(* Logix 5000 project; controller Comas_L4 vendor 1 type 14 code 193 rev 30.11; software revision 30.02; part 7 of 12 *)

        [27].Comas.Tete.Cam_Axe_Vertical[5].Master := 66.0, [27].Comas.Tete.Cam_Axe_Vertical[5].Slave := 14.0, [27].Comas.Tete.Cam_Axe_Vertical[5].SegmentType := 1, [27].Comas.Tete.Cam_Axe_Vertical[6].Master := 86.0, [27].Comas.Tete.Cam_Axe_Vertical[7].Master := 95.0, [27].Comas.Tete.Longueur_Cam_Axe_H := 8, [27].Comas.Tete.Offset_Vertical_Gauche := 38.0, [27].Comas.Tete.Offset_Horizontal_Gauche := 95.0, [27].Comas.Tete.Cam_Axe_Horizontal_Pan.B.x := 1.0, [27].Comas.Tete.Cam_Axe_Horizontal_Pan.C.x := 10.0, [27].Comas.Tete.Cam_Axe_Horizontal_Pan.C.y := 5.0, [27].Comas.Tete.Cam_Axe_Horizontal_Pan.D.x := 30.0, [27].Comas.Tete.Cam_Axe_Horizontal_Pan.D.y := 30.0, [27].Comas.Tete.Cam_Axe_Horizontal_Pan.E.x := 10.0, [27].Comas.Tete.Cam_Axe_Horizontal_Pan.E.y := 5.0, [27].Comas.Tete.Cam_Axe_Horizontal_Pan.F.x := 10.0, [27].Comas.Tete.Cam_Axe_Horizontal_Pan.G.x := 10.0, [27].Comas.Tete.Cam_Axe_Horizontal_Pan.G.y := -10.0, [27].Comas.Tete.Cam_Axe_Vertical_Pan.K.y := 2.0, [27].Comas.Tete.Cam_Axe_Vertical_Pan.L.x := 14.0, [27].Comas.Tete.Cam_Axe_Vertical_Pan.L.y := 15.0, [27].Comas.Tete.Cam_Axe_Vertical_Pan.M.x := 5.0, [27].Comas.Tete.Cam_Axe_Vertical_Pan.M.y := 14.0, [27].Comas.Tete.Cam_Axe_Vertical_Pan.N.x := 15.0, [27].Comas.Tete.Offset_Vertical_Droit := 45.0, [27].Comas.Tete.Offset_Horizontal_Droit := 95.0, [27].Comas.Pompe.Start_Cam_Logique_Avance := 1.0, [27].Comas.Pompe.Stop_Cam_Logique_Avance := 14.0, [27].Comas.Pompe.Start_Cam_Logique_Recul := 16.0, [27].Comas.Pompe.Stop_Cam_Logique_Recul := 31.0, [27].Comas.Pompe.Consigne_Vitesse_Avance := 13.2, [27].Comas.Pompe.Consigne_Acc_Dec_Avance := 40.0, [27].Comas.Pompe.Consigne_Jerk_Avance := 100.0, [27].Comas.Pompe.Consigne_Acc_Dec_Recul := 40.0, [27].Comas.Pompe.Consigne_Jerk_Recul := 100.0, [27].Comas.Pompe.Points_Pan.O.x := -10.0, [27].Comas.Pompe.Points_Pan.Q.x := 13.0, [27].Comas.Pompe.Points_Pan.S.x := -25.0, [27].Comas.Pompe.Points_Pan.U.x := 15.0, [27].Comas.Pompe.Reserve_Bool1 := 1, [27].Comas.Rouleaux.Syncho_Pompe := 1, [27].Comas.Rouleaux.Consigne_Vitesse := 30.0, [27].Comas.Rouleaux.Consigne_Acc_Dec := 40.0, [27].Comas.Rouleaux.Consigne_Jerk := 100.0, [27].Comas.Rouleaux.Reserve_Real1 := -20.0, [27].Comas.Coupe_Fil.Activation := 1, [27].Comas.Coupe_Fil.Start_Cam_Logique_Virtuelle := 11.0, [27].Comas.Coupe_Fil.Stop_Cam_Logique_Virtuelle := 21.0, [27].Comas.Coupe_Fil.Consigne_Vitesse_Virtuelle := 250.0, [27].Comas.Coupe_Fil.Consigne_Acc_Dec_Virtuelle := 1000.0, [27].Comas.Coupe_Fil.Consigne_Jerk_Virtuelle := 50.0, [27].Comas.Coupe_Fil.Cam_Axe[0].SegmentType := 1, [27].Comas.Coupe_Fil.Cam_Axe[1].Master := 180.0, [27].Comas.Coupe_Fil.Cam_Axe[1].Slave := 180.0, [27].Comas.Coupe_Fil.Cam_Axe[2].Master := 250.0, [27].Comas.Coupe_Fil.Cam_Axe[2].Slave := 200.0, [27].Comas.Coupe_Fil.Cam_Axe[2].SegmentType := 1, [27].Comas.Coupe_Fil.Cam_Axe[3].Master := 360.0, [27].Comas.Coupe_Fil.Cam_Axe[3].Slave := 360.0, [27].Comas.Coupe_Fil.Cam_Axe[3].SegmentType := 1,
        [27].Comas.Coupe_Fil.Cam_Axe[4].SegmentType := 1, [27].Comas.Coupe_Fil.Points_Pan.W.x := -40.0, [27].Comas.Coupe_Fil.Reserve_Bool1 := 1, [27].Comas.Consigne_Vitesse_Manu_mm := 2.0, [27].Comas.Consigne_Acc_Decc_Manu_mm := 10.0, [27].Comas.Consigne_Jerk_Manu := 100.0, [27].Comas.Activation_Cam_Auto := 1, [27].Comas.Distance_CPT_Presence_Produit := 520, [27].Comas.Consigne_Vitesse_Manu_Tour := 10.0, [27].Comas.Consigne_Acc_Decc_Manu_Tour := 10.0, [27].Comas.Mode_Decoreuse_Cam_Logique := 1, [27].Comas.Reserve_Real3 := 1.0, [27].Comas.Reserve_Real4 := 1.0, [27].Comas.Reserve_Real5 := 5.0, [27].Comas.Reserve_Real6 := 200.0, [27].Reserve_Real2 := 200.0, [27].Reserve_Real3 := 10.0, [28].Name := 'Galette framboise', [28].Comas.Pas_Machine := 78, [28].Comas.Came_Maitre[1].Master := 78.0, [28].Comas.Came_Maitre[1].Slave := 78.0, [28].Comas.Longueur_Came_Maitre := 2, [28].Comas.Tete.Stop_Cam_Logique_Degagement := 10.0, [28].Comas.Tete.Position_Degagement_H := 50.0, [28].Comas.Tete.Position_Degagement_V := 37.0, [28].Comas.Tete.Hauteur_Tete := -23, [28].Comas.Tete.Cam_Axe_Horizontal[1].Master := 1.0, [28].Comas.Tete.Cam_Axe_Horizontal[2].Master := 11.0, [28].Comas.Tete.Cam_Axe_Horizontal[2].Slave := -3.0, [28].Comas.Tete.Cam_Axe_Horizontal[3].Master := 41.0, [28].Comas.Tete.Cam_Axe_Horizontal[3].Slave := -6.0, [28].Comas.Tete.Cam_Axe_Horizontal[3].SegmentType := 1, [28].Comas.Tete.Cam_Axe_Horizontal[4].Master := 53.0, [28].Comas.Tete.Cam_Axe_Horizontal[4].Slave := 4.0, [28].Comas.Tete.Cam_Axe_Horizontal[4].SegmentType := 1, [28].Comas.Tete.Cam_Axe_Horizontal[5].Master := 63.0, [28].Comas.Tete.Cam_Axe_Horizontal[5].Slave := 9.0, [28].Comas.Tete.Cam_Axe_Horizontal[5].SegmentType := 1, [28].Comas.Tete.Cam_Axe_Horizontal[6].Master := 73.0, [28].Comas.Tete.Cam_Axe_Horizontal[6].Slave := 4.0, [28].Comas.Tete.Cam_Axe_Horizontal[6].SegmentType := 1, [28].Comas.Tete.Cam_Axe_Horizontal[7].Master := 78.0, [28].Comas.Tete.Cam_Axe_Vertical[1].Master := 1.0, [28].Comas.Tete.Cam_Axe_Vertical[2].Master := 11.0, [28].Comas.Tete.Cam_Axe_Vertical[3].Master := 41.0, [28].Comas.Tete.Cam_Axe_Vertical[3].SegmentType := 1, [28].Comas.Tete.Cam_Axe_Vertical[4].Master := 53.0, [28].Comas.Tete.Cam_Axe_Vertical[4].Slave := 15.0, [28].Comas.Tete.Cam_Axe_Vertical[5].Master := 63.0, [28].Comas.Tete.Cam_Axe_Vertical[5].Slave := 20.0, [28].Comas.Tete.Cam_Axe_Vertical[5].SegmentType := 1, [28].Comas.Tete.Cam_Axe_Vertical[6].Master := 73.0, [28].Comas.Tete.Cam_Axe_Vertical[6].Slave := 12.0, [28].Comas.Tete.Cam_Axe_Vertical[6].SegmentType := 1, [28].Comas.Tete.Cam_Axe_Vertical[7].Master := 78.0, [28].Comas.Tete.Longueur_Cam_Axe_H := 8, [28].Comas.Tete.Offset_Vertical_Gauche := 38.0, [28].Comas.Tete.Offset_Horizontal_Gauche := 94.0, [28].Comas.Tete.Cam_Axe_Horizontal_Pan.B.x := 1.0, [28].Comas.Tete.Cam_Axe_Horizontal_Pan.C.x := 10.0,
        [28].Comas.Tete.Cam_Axe_Horizontal_Pan.C.y := -3.0, [28].Comas.Tete.Cam_Axe_Horizontal_Pan.D.x := 30.0, [28].Comas.Tete.Cam_Axe_Horizontal_Pan.D.y := 5.0, [28].Comas.Tete.Cam_Axe_Horizontal_Pan.E.x := 12.0, [28].Comas.Tete.Cam_Axe_Horizontal_Pan.E.y := 10.0, [28].Comas.Tete.Cam_Axe_Horizontal_Pan.F.x := 10.0, [28].Comas.Tete.Cam_Axe_Horizontal_Pan.F.y := 5.0, [28].Comas.Tete.Cam_Axe_Horizontal_Pan.G.x := 10.0, [28].Comas.Tete.Cam_Axe_Horizontal_Pan.G.y := -5.0, [28].Comas.Tete.Cam_Axe_Vertical_Pan.L.y := 15.0, [28].Comas.Tete.Cam_Axe_Vertical_Pan.M.y := 20.0, [28].Comas.Tete.Cam_Axe_Vertical_Pan.N.y := 12.0, [28].Comas.Tete.Offset_Vertical_Droit := 45.0, [28].Comas.Tete.Offset_Horizontal_Droit := 94.0, [28].Comas.Tete.Reserve_Real1 := -8.0, [28].Comas.Pompe.Start_Cam_Logique_Avance := 1.0, [28].Comas.Pompe.Stop_Cam_Logique_Avance := 14.0, [28].Comas.Pompe.Start_Cam_Logique_Recul := 41.0, [28].Comas.Pompe.Stop_Cam_Logique_Recul := 41.0, [28].Comas.Pompe.Consigne_Vitesse_Avance := 18.2, [28].Comas.Pompe.Consigne_Acc_Dec_Avance := 40.0, [28].Comas.Pompe.Consigne_Jerk_Avance := 100.0, [28].Comas.Pompe.Consigne_Acc_Dec_Recul := 40.0, [28].Comas.Pompe.Consigne_Jerk_Recul := 100.0, [28].Comas.Pompe.Points_Pan.O.x := -10.0, [28].Comas.Pompe.Points_Pan.Q.x := 13.0, [28].Comas.Pompe.Reserve_Bool1 := 1, [28].Comas.Rouleaux.Syncho_Pompe := 1, [28].Comas.Rouleaux.Consigne_Vitesse := 25.0, [28].Comas.Rouleaux.Consigne_Acc_Dec := 40.0, [28].Comas.Rouleaux.Consigne_Jerk := 100.0, [28].Comas.Rouleaux.Reserve_Real1 := -10.0, [28].Comas.Coupe_Fil.Activation := 1, [28].Comas.Coupe_Fil.Start_Cam_Logique_Virtuelle := 18.0, [28].Comas.Coupe_Fil.Stop_Cam_Logique_Virtuelle := 28.0, [28].Comas.Coupe_Fil.Consigne_Vitesse_Virtuelle := 400.0, [28].Comas.Coupe_Fil.Consigne_Acc_Dec_Virtuelle := 1200.0, [28].Comas.Coupe_Fil.Consigne_Jerk_Virtuelle := 50.0, [28].Comas.Coupe_Fil.Cam_Axe[0].SegmentType := 1, [28].Comas.Coupe_Fil.Cam_Axe[1].Master := 180.0, [28].Comas.Coupe_Fil.Cam_Axe[1].Slave := 180.0, [28].Comas.Coupe_Fil.Cam_Axe[2].Master := 250.0, [28].Comas.Coupe_Fil.Cam_Axe[2].Slave := 200.0, [28].Comas.Coupe_Fil.Cam_Axe[2].SegmentType := 1, [28].Comas.Coupe_Fil.Cam_Axe[3].Master := 360.0, [28].Comas.Coupe_Fil.Cam_Axe[3].Slave := 360.0, [28].Comas.Coupe_Fil.Cam_Axe[3].SegmentType := 1, [28].Comas.Coupe_Fil.Cam_Axe[4].SegmentType := 1, [28].Comas.Coupe_Fil.Points_Pan.W.x := -35.0, [28].Comas.Coupe_Fil.Reserve_Bool1 := 1, [28].Comas.Consigne_Vitesse_Manu_mm := 2.0, [28].Comas.Consigne_Acc_Decc_Manu_mm := 10.0, [28].Comas.Consigne_Jerk_Manu := 100.0, [28].Comas.Activation_Cam_Auto := 1, [28].Comas.Distance_CPT_Presence_Produit := 520, [28].Comas.Consigne_Vitesse_Manu_Tour := 10.0, [28].Comas.Consigne_Acc_Decc_Manu_Tour := 10.0, [28].Comas.Mode_Decoreuse_Cam_Logique := 1, [28].Comas.Reserve_Real3 := 1.0, [28].Comas.Reserve_Real4 := 1.0,
        [28].Comas.Reserve_Real5 := 5.0, [28].Comas.Reserve_Real6 := 200.0, [28].Reserve_Real2 := 200.0, [28].Reserve_Real3 := 10.0, [29].Name := 'Galette orange', [29].Comas.Pas_Machine := 78, [29].Comas.Came_Maitre[1].Master := 78.0, [29].Comas.Came_Maitre[1].Slave := 78.0, [29].Comas.Longueur_Came_Maitre := 2, [29].Comas.Tete.Stop_Cam_Logique_Degagement := 10.0, [29].Comas.Tete.Position_Degagement_H := 50.0, [29].Comas.Tete.Position_Degagement_V := 37.0, [29].Comas.Tete.Hauteur_Tete := -24, [29].Comas.Tete.Cam_Axe_Horizontal[1].Master := 1.0, [29].Comas.Tete.Cam_Axe_Horizontal[2].Master := 11.0, [29].Comas.Tete.Cam_Axe_Horizontal[2].Slave := -3.0, [29].Comas.Tete.Cam_Axe_Horizontal[3].Master := 41.0, [29].Comas.Tete.Cam_Axe_Horizontal[3].Slave := -6.0, [29].Comas.Tete.Cam_Axe_Horizontal[3].SegmentType := 1, [29].Comas.Tete.Cam_Axe_Horizontal[4].Master := 53.0, [29].Comas.Tete.Cam_Axe_Horizontal[4].Slave := 4.0, [29].Comas.Tete.Cam_Axe_Horizontal[4].SegmentType := 1, [29].Comas.Tete.Cam_Axe_Horizontal[5].Master := 63.0, [29].Comas.Tete.Cam_Axe_Horizontal[5].Slave := 9.0, [29].Comas.Tete.Cam_Axe_Horizontal[5].SegmentType := 1, [29].Comas.Tete.Cam_Axe_Horizontal[6].Master := 73.0, [29].Comas.Tete.Cam_Axe_Horizontal[6].Slave := 4.0, [29].Comas.Tete.Cam_Axe_Horizontal[6].SegmentType := 1, [29].Comas.Tete.Cam_Axe_Horizontal[7].Master := 78.0, [29].Comas.Tete.Cam_Axe_Vertical[1].Master := 1.0, [29].Comas.Tete.Cam_Axe_Vertical[2].Master := 11.0, [29].Comas.Tete.Cam_Axe_Vertical[3].Master := 41.0, [29].Comas.Tete.Cam_Axe_Vertical[3].SegmentType := 1, [29].Comas.Tete.Cam_Axe_Vertical[4].Master := 53.0, [29].Comas.Tete.Cam_Axe_Vertical[4].Slave := 15.0, [29].Comas.Tete.Cam_Axe_Vertical[5].Master := 63.0, [29].Comas.Tete.Cam_Axe_Vertical[5].Slave := 25.0, [29].Comas.Tete.Cam_Axe_Vertical[5].SegmentType := 1, [29].Comas.Tete.Cam_Axe_Vertical[6].Master := 73.0, [29].Comas.Tete.Cam_Axe_Vertical[6].Slave := 12.0, [29].Comas.Tete.Cam_Axe_Vertical[6].SegmentType := 1, [29].Comas.Tete.Cam_Axe_Vertical[7].Master := 78.0, [29].Comas.Tete.Longueur_Cam_Axe_H := 8, [29].Comas.Tete.Offset_Vertical_Gauche := 38.0, [29].Comas.Tete.Offset_Horizontal_Gauche := 94.0, [29].Comas.Tete.Cam_Axe_Horizontal_Pan.B.x := 1.0, [29].Comas.Tete.Cam_Axe_Horizontal_Pan.C.x := 10.0, [29].Comas.Tete.Cam_Axe_Horizontal_Pan.C.y := -3.0, [29].Comas.Tete.Cam_Axe_Horizontal_Pan.D.x := 30.0, [29].Comas.Tete.Cam_Axe_Horizontal_Pan.D.y := 5.0, [29].Comas.Tete.Cam_Axe_Horizontal_Pan.E.x := 12.0, [29].Comas.Tete.Cam_Axe_Horizontal_Pan.E.y := 10.0, [29].Comas.Tete.Cam_Axe_Horizontal_Pan.F.x := 10.0, [29].Comas.Tete.Cam_Axe_Horizontal_Pan.F.y := 5.0, [29].Comas.Tete.Cam_Axe_Horizontal_Pan.G.x := 10.0, [29].Comas.Tete.Cam_Axe_Horizontal_Pan.G.y := -5.0, [29].Comas.Tete.Cam_Axe_Vertical_Pan.L.y := 15.0, [29].Comas.Tete.Cam_Axe_Vertical_Pan.M.y := 25.0, [29].Comas.Tete.Cam_Axe_Vertical_Pan.N.y := 12.0, [29].Comas.Tete.Offset_Vertical_Droit := 45.0,
        [29].Comas.Tete.Offset_Horizontal_Droit := 94.0, [29].Comas.Tete.Reserve_Real1 := -8.0, [29].Comas.Pompe.Start_Cam_Logique_Avance := 16.0, [29].Comas.Pompe.Stop_Cam_Logique_Avance := 29.0, [29].Comas.Pompe.Start_Cam_Logique_Recul := 41.0, [29].Comas.Pompe.Stop_Cam_Logique_Recul := 41.0, [29].Comas.Pompe.Consigne_Vitesse_Avance := 21.6, [29].Comas.Pompe.Consigne_Acc_Dec_Avance := 40.0, [29].Comas.Pompe.Consigne_Jerk_Avance := 100.0, [29].Comas.Pompe.Consigne_Acc_Dec_Recul := 40.0, [29].Comas.Pompe.Consigne_Jerk_Recul := 100.0, [29].Comas.Pompe.Points_Pan.O.x := 5.0, [29].Comas.Pompe.Points_Pan.Q.x := 13.0, [29].Comas.Pompe.Reserve_Bool1 := 1, [29].Comas.Rouleaux.Syncho_Pompe := 1, [29].Comas.Rouleaux.Consigne_Vitesse := 26.0, [29].Comas.Rouleaux.Consigne_Acc_Dec := 40.0, [29].Comas.Rouleaux.Consigne_Jerk := 100.0, [29].Comas.Rouleaux.Reserve_Real1 := -20.0, [29].Comas.Coupe_Fil.Activation := 1, [29].Comas.Coupe_Fil.Start_Cam_Logique_Virtuelle := 18.0, [29].Comas.Coupe_Fil.Stop_Cam_Logique_Virtuelle := 28.0, [29].Comas.Coupe_Fil.Consigne_Vitesse_Virtuelle := 380.0, [29].Comas.Coupe_Fil.Consigne_Acc_Dec_Virtuelle := 1200.0, [29].Comas.Coupe_Fil.Consigne_Jerk_Virtuelle := 50.0, [29].Comas.Coupe_Fil.Cam_Axe[0].SegmentType := 1, [29].Comas.Coupe_Fil.Cam_Axe[1].Master := 180.0, [29].Comas.Coupe_Fil.Cam_Axe[1].Slave := 180.0, [29].Comas.Coupe_Fil.Cam_Axe[2].Master := 250.0, [29].Comas.Coupe_Fil.Cam_Axe[2].Slave := 200.0, [29].Comas.Coupe_Fil.Cam_Axe[2].SegmentType := 1, [29].Comas.Coupe_Fil.Cam_Axe[3].Master := 360.0, [29].Comas.Coupe_Fil.Cam_Axe[3].Slave := 360.0, [29].Comas.Coupe_Fil.Cam_Axe[3].SegmentType := 1, [29].Comas.Coupe_Fil.Cam_Axe[4].SegmentType := 1, [29].Comas.Coupe_Fil.Points_Pan.W.x := -35.0, [29].Comas.Coupe_Fil.Reserve_Bool1 := 1, [29].Comas.Consigne_Vitesse_Manu_mm := 2.0, [29].Comas.Consigne_Acc_Decc_Manu_mm := 10.0, [29].Comas.Consigne_Jerk_Manu := 100.0, [29].Comas.Activation_Cam_Auto := 1, [29].Comas.Distance_CPT_Presence_Produit := 520, [29].Comas.Consigne_Vitesse_Manu_Tour := 10.0, [29].Comas.Consigne_Acc_Decc_Manu_Tour := 10.0, [29].Comas.Mode_Decoreuse_Cam_Logique := 1, [29].Comas.Reserve_Real3 := 1.0, [29].Comas.Reserve_Real4 := 1.0, [29].Comas.Reserve_Real5 := 5.0, [29].Comas.Reserve_Real6 := 200.0, [29].Reserve_Real2 := 200.0, [29].Reserve_Real3 := 10.0, [30].Name := 'ROCHER 44', [30].Comas.Pas_Machine := 78, [30].Comas.Came_Maitre[1].Master := 78.0, [30].Comas.Came_Maitre[1].Slave := 78.0, [30].Comas.Longueur_Came_Maitre := 2, [30].Comas.Tete.Stop_Cam_Logique_Degagement := 10.0, [30].Comas.Tete.Position_Degagement_H := 50.0, [30].Comas.Tete.Position_Degagement_V := 35.0, [30].Comas.Tete.Hauteur_Tete := -1,
        [30].Comas.Tete.Cam_Axe_Horizontal[1].Master := 1.0, [30].Comas.Tete.Cam_Axe_Horizontal[1].SegmentType := 1, [30].Comas.Tete.Cam_Axe_Horizontal[2].Master := 6.0, [30].Comas.Tete.Cam_Axe_Horizontal[2].Slave := 2.0, [30].Comas.Tete.Cam_Axe_Horizontal[3].Master := 31.0, [30].Comas.Tete.Cam_Axe_Horizontal[3].Slave := 30.0, [30].Comas.Tete.Cam_Axe_Horizontal[3].SegmentType := 1, [30].Comas.Tete.Cam_Axe_Horizontal[4].Master := 46.0, [30].Comas.Tete.Cam_Axe_Horizontal[4].Slave := 50.0, [30].Comas.Tete.Cam_Axe_Horizontal[5].Master := 51.0, [30].Comas.Tete.Cam_Axe_Horizontal[5].Slave := 50.0, [30].Comas.Tete.Cam_Axe_Horizontal[5].SegmentType := 1, [30].Comas.Tete.Cam_Axe_Horizontal[6].Master := 61.0, [30].Comas.Tete.Cam_Axe_Horizontal[6].Slave := 40.0, [30].Comas.Tete.Cam_Axe_Horizontal[6].SegmentType := 1, [30].Comas.Tete.Cam_Axe_Horizontal[7].Master := 78.0, [30].Comas.Tete.Cam_Axe_Vertical[1].Master := 1.0, [30].Comas.Tete.Cam_Axe_Vertical[2].Master := 6.0, [30].Comas.Tete.Cam_Axe_Vertical[3].Master := 21.0, [30].Comas.Tete.Cam_Axe_Vertical[3].SegmentType := 1, [30].Comas.Tete.Cam_Axe_Vertical[4].Master := 46.0, [30].Comas.Tete.Cam_Axe_Vertical[4].Slave := 5.0, [30].Comas.Tete.Cam_Axe_Vertical[5].Master := 56.0, [30].Comas.Tete.Cam_Axe_Vertical[5].Slave := 10.0, [30].Comas.Tete.Cam_Axe_Vertical[5].SegmentType := 1, [30].Comas.Tete.Cam_Axe_Vertical[6].Master := 71.0, [30].Comas.Tete.Cam_Axe_Vertical[7].Master := 78.0, [30].Comas.Tete.Longueur_Cam_Axe_H := 8, [30].Comas.Tete.Offset_Vertical_Gauche := 38.0, [30].Comas.Tete.Offset_Horizontal_Gauche := 95.0, [30].Comas.Tete.Cam_Axe_Horizontal_Pan.B.x := 1.0, [30].Comas.Tete.Cam_Axe_Horizontal_Pan.C.x := 5.0, [30].Comas.Tete.Cam_Axe_Horizontal_Pan.C.y := 2.0, [30].Comas.Tete.Cam_Axe_Horizontal_Pan.D.x := 25.0, [30].Comas.Tete.Cam_Axe_Horizontal_Pan.D.y := 28.0, [30].Comas.Tete.Cam_Axe_Horizontal_Pan.E.x := 15.0, [30].Comas.Tete.Cam_Axe_Horizontal_Pan.E.y := 20.0, [30].Comas.Tete.Cam_Axe_Horizontal_Pan.F.x := 5.0, [30].Comas.Tete.Cam_Axe_Horizontal_Pan.G.x := 10.0, [30].Comas.Tete.Cam_Axe_Horizontal_Pan.G.y := -10.0, [30].Comas.Tete.Cam_Axe_Vertical_Pan.K.x := -10.0, [30].Comas.Tete.Cam_Axe_Vertical_Pan.L.y := 5.0, [30].Comas.Tete.Cam_Axe_Vertical_Pan.M.x := 5.0, [30].Comas.Tete.Cam_Axe_Vertical_Pan.M.y := 10.0, [30].Comas.Tete.Cam_Axe_Vertical_Pan.N.x := 10.0, [30].Comas.Tete.Offset_Vertical_Droit := 45.0, [30].Comas.Tete.Offset_Horizontal_Droit := 95.0, [30].Comas.Pompe.Start_Cam_Logique_Avance := -14.0, [30].Comas.Pompe.Stop_Cam_Logique_Avance := 16.0, [30].Comas.Pompe.Start_Cam_Logique_Recul := 22.0, [30].Comas.Pompe.Stop_Cam_Logique_Recul := 43.0, [30].Comas.Pompe.Consigne_Vitesse_Avance := 17.3, [30].Comas.Pompe.Consigne_Acc_Dec_Avance := 40.0, [30].Comas.Pompe.Consigne_Jerk_Avance := 100.0, [30].Comas.Pompe.Consigne_Vitesse_Recul := -10.0, [30].Comas.Pompe.Consigne_Acc_Dec_Recul := 40.0, [30].Comas.Pompe.Consigne_Jerk_Recul := 100.0, [30].Comas.Pompe.Points_Pan.O.x := -20.0, [30].Comas.Pompe.Points_Pan.Q.x := 30.0, [30].Comas.Pompe.Points_Pan.S.x := 1.0,
        [30].Comas.Pompe.Points_Pan.U.x := 21.0, [30].Comas.Pompe.Reserve_Bool1 := 1, [30].Comas.Rouleaux.Syncho_Pompe := 1, [30].Comas.Rouleaux.Consigne_Vitesse := 10.0, [30].Comas.Rouleaux.Consigne_Acc_Dec := 40.0, [30].Comas.Rouleaux.Consigne_Jerk := 100.0, [30].Comas.Coupe_Fil.Start_Cam_Logique_Virtuelle := 11.0, [30].Comas.Coupe_Fil.Stop_Cam_Logique_Virtuelle := 21.0, [30].Comas.Coupe_Fil.Consigne_Vitesse_Virtuelle := 200.0, [30].Comas.Coupe_Fil.Consigne_Acc_Dec_Virtuelle := 1000.0, [30].Comas.Coupe_Fil.Consigne_Jerk_Virtuelle := 50.0, [30].Comas.Coupe_Fil.Cam_Axe[0].SegmentType := 1, [30].Comas.Coupe_Fil.Cam_Axe[1].Master := 180.0, [30].Comas.Coupe_Fil.Cam_Axe[1].Slave := 90.0, [30].Comas.Coupe_Fil.Cam_Axe[2].Master := 360.0, [30].Comas.Coupe_Fil.Cam_Axe[2].Slave := 360.0, [30].Comas.Coupe_Fil.Cam_Axe[2].SegmentType := 1, [30].Comas.Coupe_Fil.Points_Pan.W.x := 30.0, [30].Comas.Consigne_Vitesse_Manu_mm := 4.0, [30].Comas.Consigne_Acc_Decc_Manu_mm := 10.0, [30].Comas.Consigne_Jerk_Manu := 100.0, [30].Comas.Activation_Cam_Auto := 1, [30].Comas.Distance_CPT_Presence_Produit := 520, [30].Comas.Consigne_Vitesse_Manu_Tour := 10.0, [30].Comas.Consigne_Acc_Decc_Manu_Tour := 10.0, [30].Comas.Mode_Decoreuse_Cam_Logique := 1, [30].Comas.Reserve_Real6 := 200.0, [31].Name := 'BISC SES TOURN', [31].Comas.Pas_Machine := 84, [31].Comas.Came_Maitre[1].Master := 84.0, [31].Comas.Came_Maitre[1].Slave := 84.0, [31].Comas.Longueur_Came_Maitre := 2, [31].Comas.Tete.Stop_Cam_Logique_Degagement := 10.0, [31].Comas.Tete.Position_Degagement_H := 50.0, [31].Comas.Tete.Position_Degagement_V := 35.0, [31].Comas.Tete.Hauteur_Tete := -2, [31].Comas.Tete.Cam_Axe_Horizontal[1].Master := 16.0, [31].Comas.Tete.Cam_Axe_Horizontal[1].Slave := 11.0, [31].Comas.Tete.Cam_Axe_Horizontal[1].SegmentType := 1, [31].Comas.Tete.Cam_Axe_Horizontal[2].Master := 19.0, [31].Comas.Tete.Cam_Axe_Horizontal[2].Slave := 12.0, [31].Comas.Tete.Cam_Axe_Horizontal[3].Master := 55.0, [31].Comas.Tete.Cam_Axe_Horizontal[3].SegmentType := 1, [31].Comas.Tete.Cam_Axe_Horizontal[4].Master := 59.0, [31].Comas.Tete.Cam_Axe_Horizontal[4].Slave := -3.0, [31].Comas.Tete.Cam_Axe_Horizontal[4].SegmentType := 1, [31].Comas.Tete.Cam_Axe_Horizontal[5].Master := 69.0, [31].Comas.Tete.Cam_Axe_Horizontal[5].Slave := -3.0, [31].Comas.Tete.Cam_Axe_Horizontal[5].SegmentType := 1, [31].Comas.Tete.Cam_Axe_Horizontal[6].Master := 79.0, [31].Comas.Tete.Cam_Axe_Horizontal[6].Slave := -3.0, [31].Comas.Tete.Cam_Axe_Horizontal[6].SegmentType := 1, [31].Comas.Tete.Cam_Axe_Horizontal[7].Master := 84.0, [31].Comas.Tete.Cam_Axe_Vertical[1].Master := 10.0, [31].Comas.Tete.Cam_Axe_Vertical[1].Slave := 5.0, [31].Comas.Tete.Cam_Axe_Vertical[1].SegmentType := 1, [31].Comas.Tete.Cam_Axe_Vertical[2].Master := 19.0, [31].Comas.Tete.Cam_Axe_Vertical[2].Slave := 7.0, [31].Comas.Tete.Cam_Axe_Vertical[2].SegmentType := 1, [31].Comas.Tete.Cam_Axe_Vertical[3].Master := 53.0,
        [31].Comas.Tete.Cam_Axe_Vertical[3].SegmentType := 1, [31].Comas.Tete.Cam_Axe_Vertical[4].Master := 59.0, [31].Comas.Tete.Cam_Axe_Vertical[5].Master := 69.0, [31].Comas.Tete.Cam_Axe_Vertical[5].SegmentType := 1, [31].Comas.Tete.Cam_Axe_Vertical[6].Master := 79.0, [31].Comas.Tete.Cam_Axe_Vertical[7].Master := 84.0, [31].Comas.Tete.Longueur_Cam_Axe_H := 8, [31].Comas.Tete.Offset_Vertical_Gauche := 45.0, [31].Comas.Tete.Offset_Horizontal_Gauche := 95.0, [31].Comas.Tete.Cam_Axe_Horizontal_Pan.B.x := 16.0, [31].Comas.Tete.Cam_Axe_Horizontal_Pan.B.y := 11.0, [31].Comas.Tete.Cam_Axe_Horizontal_Pan.C.x := 3.0, [31].Comas.Tete.Cam_Axe_Horizontal_Pan.C.y := 1.0, [31].Comas.Tete.Cam_Axe_Horizontal_Pan.D.x := 36.0, [31].Comas.Tete.Cam_Axe_Horizontal_Pan.D.y := -10.0, [31].Comas.Tete.Cam_Axe_Horizontal_Pan.E.x := 4.0, [31].Comas.Tete.Cam_Axe_Horizontal_Pan.E.y := -3.0, [31].Comas.Tete.Cam_Axe_Horizontal_Pan.F.x := 10.0, [31].Comas.Tete.Cam_Axe_Horizontal_Pan.G.x := 10.0, [31].Comas.Tete.Cam_Axe_Vertical_Pan.I.x := -6.0, [31].Comas.Tete.Cam_Axe_Vertical_Pan.I.y := 5.0, [31].Comas.Tete.Cam_Axe_Vertical_Pan.J.y := 7.0, [31].Comas.Tete.Cam_Axe_Vertical_Pan.K.x := -2.0, [31].Comas.Tete.Offset_Vertical_Droit := 45.0, [31].Comas.Tete.Offset_Horizontal_Droit := 95.0, [31].Comas.Tete.Reserve_Real1 := -2.0, [31].Comas.Pompe.Start_Cam_Logique_Avance := 23.0, [31].Comas.Pompe.Stop_Cam_Logique_Avance := 50.0, [31].Comas.Pompe.Start_Cam_Logique_Recul := 54.0, [31].Comas.Pompe.Stop_Cam_Logique_Recul := 64.0, [31].Comas.Pompe.Consigne_Vitesse_Avance := 20.8, [31].Comas.Pompe.Consigne_Acc_Dec_Avance := 40.0, [31].Comas.Pompe.Consigne_Jerk_Avance := 100.0, [31].Comas.Pompe.Consigne_Acc_Dec_Recul := 40.0, [31].Comas.Pompe.Consigne_Jerk_Recul := 100.0, [31].Comas.Pompe.Points_Pan.O.x := 4.0, [31].Comas.Pompe.Points_Pan.Q.x := 27.0, [31].Comas.Pompe.Points_Pan.S.x := 1.0, [31].Comas.Pompe.Points_Pan.U.x := 10.0, [31].Comas.Pompe.Reserve_Bool1 := 1, [31].Comas.Rouleaux.Consigne_Vitesse := 25.0, [31].Comas.Rouleaux.Consigne_Acc_Dec := 40.0, [31].Comas.Rouleaux.Consigne_Jerk := 100.0, [31].Comas.Coupe_Fil.Activation := 1, [31].Comas.Coupe_Fil.Start_Cam_Logique_Virtuelle := 61.0, [31].Comas.Coupe_Fil.Stop_Cam_Logique_Virtuelle := 71.0, [31].Comas.Coupe_Fil.Consigne_Vitesse_Virtuelle := 330.0, [31].Comas.Coupe_Fil.Consigne_Acc_Dec_Virtuelle := 750.0, [31].Comas.Coupe_Fil.Consigne_Jerk_Virtuelle := 50.0, [31].Comas.Coupe_Fil.Cam_Axe[0].SegmentType := 1, [31].Comas.Coupe_Fil.Cam_Axe[1].Master := 180.0, [31].Comas.Coupe_Fil.Cam_Axe[1].Slave := 165.0, [31].Comas.Coupe_Fil.Cam_Axe[2].Master := 210.0, [31].Comas.Coupe_Fil.Cam_Axe[2].Slave := 165.0, [31].Comas.Coupe_Fil.Cam_Axe[2].SegmentType := 1, [31].Comas.Coupe_Fil.Cam_Axe[3].Master := 250.0, [31].Comas.Coupe_Fil.Cam_Axe[3].Slave := 250.0, [31].Comas.Coupe_Fil.Cam_Axe[3].SegmentType := 1, [31].Comas.Coupe_Fil.Cam_Axe[4].Master := 360.0, [31].Comas.Coupe_Fil.Cam_Axe[4].Slave := 360.0,
        [31].Comas.Coupe_Fil.Cam_Axe[4].SegmentType := 1, [31].Comas.Coupe_Fil.Points_Pan.W.x := 2.0, [31].Comas.Coupe_Fil.Reserve_Bool1 := 1, [31].Comas.Consigne_Vitesse_Manu_mm := 2.0, [31].Comas.Consigne_Acc_Decc_Manu_mm := 10.0, [31].Comas.Consigne_Jerk_Manu := 100.0, [31].Comas.Activation_Cam_Auto := 1, [31].Comas.Distance_CPT_Presence_Produit := 520, [31].Comas.Consigne_Vitesse_Manu_Tour := 10.0, [31].Comas.Consigne_Acc_Decc_Manu_Tour := 10.0, [31].Comas.Mode_Decoreuse_Cam_Logique := 1, [31].Comas.Reserve_Real3 := 1.0, [31].Comas.Reserve_Real4 := 1.0, [31].Comas.Reserve_Real5 := 5.0, [31].Comas.Reserve_Real6 := 200.0, [31].Reserve_Real2 := 200.0, [31].Reserve_Real3 := 10.0, [33].Name := 'tartelette SSA', [33].Comas.Pas_Machine := 100, [33].Comas.Came_Maitre[1].Master := 100.0, [33].Comas.Came_Maitre[1].Slave := 100.0, [33].Comas.Longueur_Came_Maitre := 2, [33].Comas.Tete.Stop_Cam_Logique_Degagement := 10.0, [33].Comas.Tete.Position_Degagement_H := 20.0, [33].Comas.Tete.Position_Degagement_V := 37.0, [33].Comas.Tete.Hauteur_Tete := -18, [33].Comas.Tete.Cam_Axe_Horizontal[1].Master := 1.0, [33].Comas.Tete.Cam_Axe_Horizontal[1].Slave := 1.0, [33].Comas.Tete.Cam_Axe_Horizontal[1].SegmentType := 1, [33].Comas.Tete.Cam_Axe_Horizontal[2].Master := 9.0, [33].Comas.Tete.Cam_Axe_Horizontal[2].Slave := 16.0, [33].Comas.Tete.Cam_Axe_Horizontal[2].SegmentType := 1, [33].Comas.Tete.Cam_Axe_Horizontal[3].Master := 40.0, [33].Comas.Tete.Cam_Axe_Horizontal[3].Slave := 94.0, [33].Comas.Tete.Cam_Axe_Horizontal[3].SegmentType := 1, [33].Comas.Tete.Cam_Axe_Horizontal[4].Master := 50.0, [33].Comas.Tete.Cam_Axe_Horizontal[4].Slave := 104.0, [33].Comas.Tete.Cam_Axe_Horizontal[5].Master := 55.0, [33].Comas.Tete.Cam_Axe_Horizontal[5].Slave := 94.0, [33].Comas.Tete.Cam_Axe_Horizontal[5].SegmentType := 1, [33].Comas.Tete.Cam_Axe_Horizontal[6].Master := 65.0, [33].Comas.Tete.Cam_Axe_Horizontal[6].Slave := 69.0, [33].Comas.Tete.Cam_Axe_Horizontal[6].SegmentType := 1, [33].Comas.Tete.Cam_Axe_Horizontal[7].Master := 100.0, [33].Comas.Tete.Cam_Axe_Vertical[0].Slave := 15.0, [33].Comas.Tete.Cam_Axe_Vertical[1].Master := 1.0, [33].Comas.Tete.Cam_Axe_Vertical[1].Slave := 15.0, [33].Comas.Tete.Cam_Axe_Vertical[2].Master := 9.0, [33].Comas.Tete.Cam_Axe_Vertical[2].Slave := 10.0, [33].Comas.Tete.Cam_Axe_Vertical[3].Master := 52.0, [33].Comas.Tete.Cam_Axe_Vertical[3].Slave := 12.0, [33].Comas.Tete.Cam_Axe_Vertical[3].SegmentType := 1, [33].Comas.Tete.Cam_Axe_Vertical[4].Master := 62.0, [33].Comas.Tete.Cam_Axe_Vertical[4].Slave := 12.0, [33].Comas.Tete.Cam_Axe_Vertical[5].Master := 67.0, [33].Comas.Tete.Cam_Axe_Vertical[5].Slave := 12.0, [33].Comas.Tete.Cam_Axe_Vertical[5].SegmentType := 1, [33].Comas.Tete.Cam_Axe_Vertical[6].Master := 85.0, [33].Comas.Tete.Cam_Axe_Vertical[6].Slave := 50.0, [33].Comas.Tete.Cam_Axe_Vertical[6].SegmentType := 1,
        [33].Comas.Tete.Cam_Axe_Vertical[7].Master := 100.0, [33].Comas.Tete.Cam_Axe_Vertical[7].Slave := 15.0, [33].Comas.Tete.Longueur_Cam_Axe_H := 8, [33].Comas.Tete.Offset_Vertical_Gauche := 38.0, [33].Comas.Tete.Offset_Horizontal_Gauche := 95.0, [33].Comas.Tete.Cam_Axe_Horizontal_Pan.B.x := 1.0, [33].Comas.Tete.Cam_Axe_Horizontal_Pan.B.y := 1.0, [33].Comas.Tete.Cam_Axe_Horizontal_Pan.C.x := 8.0, [33].Comas.Tete.Cam_Axe_Horizontal_Pan.C.y := 15.0, [33].Comas.Tete.Cam_Axe_Horizontal_Pan.D.x := 31.0, [33].Comas.Tete.Cam_Axe_Horizontal_Pan.D.y := 78.0, [33].Comas.Tete.Cam_Axe_Horizontal_Pan.E.x := 10.0, [33].Comas.Tete.Cam_Axe_Horizontal_Pan.E.y := 10.0, [33].Comas.Tete.Cam_Axe_Horizontal_Pan.F.x := 5.0, [33].Comas.Tete.Cam_Axe_Horizontal_Pan.F.y := -10.0, [33].Comas.Tete.Cam_Axe_Horizontal_Pan.G.x := 10.0, [33].Comas.Tete.Cam_Axe_Horizontal_Pan.G.y := -25.0, [33].Comas.Tete.Cam_Axe_Vertical_Pan.H.y := 15.0, [33].Comas.Tete.Cam_Axe_Vertical_Pan.I.y := 15.0, [33].Comas.Tete.Cam_Axe_Vertical_Pan.J.y := 10.0, [33].Comas.Tete.Cam_Axe_Vertical_Pan.K.x := 12.0, [33].Comas.Tete.Cam_Axe_Vertical_Pan.K.y := 12.0, [33].Comas.Tete.Cam_Axe_Vertical_Pan.L.x := 12.0, [33].Comas.Tete.Cam_Axe_Vertical_Pan.L.y := 12.0, [33].Comas.Tete.Cam_Axe_Vertical_Pan.M.x := 12.0, [33].Comas.Tete.Cam_Axe_Vertical_Pan.M.y := 12.0, [33].Comas.Tete.Cam_Axe_Vertical_Pan.N.x := 20.0, [33].Comas.Tete.Cam_Axe_Vertical_Pan.N.y := 50.0, [33].Comas.Tete.Offset_Vertical_Droit := 45.0, [33].Comas.Tete.Offset_Horizontal_Droit := 95.0, [33].Comas.Pompe.Start_Cam_Logique_Avance := -6.0, [33].Comas.Pompe.Stop_Cam_Logique_Avance := 44.0, [33].Comas.Pompe.Start_Cam_Logique_Recul := 44.0, [33].Comas.Pompe.Stop_Cam_Logique_Recul := 64.0, [33].Comas.Pompe.Consigne_Vitesse_Avance := 9.5, [33].Comas.Pompe.Consigne_Acc_Dec_Avance := 40.0, [33].Comas.Pompe.Consigne_Jerk_Avance := 80.0, [33].Comas.Pompe.Consigne_Vitesse_Recul := -16.0, [33].Comas.Pompe.Consigne_Acc_Dec_Recul := 40.0, [33].Comas.Pompe.Consigne_Jerk_Recul := 100.0, [33].Comas.Pompe.Points_Pan.O.x := -15.0, [33].Comas.Pompe.Points_Pan.Q.x := 50.0, [33].Comas.Pompe.Points_Pan.S.x := -8.0, [33].Comas.Pompe.Points_Pan.U.x := 20.0, [33].Comas.Pompe.Reserve_Bool1 := 1, [33].Comas.Rouleaux.Syncho_Pompe := 1, [33].Comas.Rouleaux.Consigne_Vitesse := 15.0, [33].Comas.Rouleaux.Consigne_Acc_Dec := 40.0, [33].Comas.Rouleaux.Consigne_Jerk := 100.0, [33].Comas.Coupe_Fil.Start_Cam_Logique_Virtuelle := 11.0, [33].Comas.Coupe_Fil.Stop_Cam_Logique_Virtuelle := 21.0, [33].Comas.Coupe_Fil.Consigne_Vitesse_Virtuelle := 200.0, [33].Comas.Coupe_Fil.Consigne_Acc_Dec_Virtuelle := 1000.0, [33].Comas.Coupe_Fil.Consigne_Jerk_Virtuelle := 50.0, [33].Comas.Coupe_Fil.Cam_Axe[0].SegmentType := 1, [33].Comas.Coupe_Fil.Cam_Axe[1].Master := 180.0, [33].Comas.Coupe_Fil.Cam_Axe[1].Slave := 90.0, [33].Comas.Coupe_Fil.Cam_Axe[2].Master := 360.0, [33].Comas.Coupe_Fil.Cam_Axe[2].Slave := 360.0, [33].Comas.Coupe_Fil.Cam_Axe[2].SegmentType := 1,
        [33].Comas.Coupe_Fil.Points_Pan.W.x := 30.0, [33].Comas.Consigne_Vitesse_Manu_mm := 2.0, [33].Comas.Consigne_Acc_Decc_Manu_mm := 10.0, [33].Comas.Consigne_Jerk_Manu := 100.0, [33].Comas.Activation_Cam_Auto := 1, [33].Comas.Mode_CPT_Presence := 1, [33].Comas.Distance_CPT_Presence_Produit := 746, [33].Comas.Consigne_Vitesse_Manu_Tour := 10.0, [33].Comas.Consigne_Acc_Decc_Manu_Tour := 10.0, [33].Comas.Mode_Decoreuse_Cam_Logique := 1, [33].Comas.Reserve_Real1 := 23.0, [33].Comas.Reserve_Real3 := 1.0, [33].Comas.Reserve_Real4 := 1.0, [33].Comas.Reserve_Real5 := 5.0, [33].Comas.Reserve_Real6 := 200.0, [33].Reserve_Real2 := 200.0, [33].Reserve_Real3 := 10.0, [34].Name := 'terra', [34].Comas.Pas_Machine := 94, [34].Comas.Came_Maitre[1].Master := 94.0, [34].Comas.Came_Maitre[1].Slave := 94.0, [34].Comas.Longueur_Came_Maitre := 2, [34].Comas.Tete.Stop_Cam_Logique_Degagement := 10.0, [34].Comas.Tete.Position_Degagement_H := 50.0, [34].Comas.Tete.Position_Degagement_V := 37.0, [34].Comas.Tete.Hauteur_Tete := -3, [34].Comas.Tete.Cam_Axe_Horizontal[1].Master := 1.0, [34].Comas.Tete.Cam_Axe_Horizontal[1].SegmentType := 1, [34].Comas.Tete.Cam_Axe_Horizontal[2].Master := 11.0, [34].Comas.Tete.Cam_Axe_Horizontal[2].Slave := 10.0, [34].Comas.Tete.Cam_Axe_Horizontal[3].Master := 41.0, [34].Comas.Tete.Cam_Axe_Horizontal[3].Slave := 35.0, [34].Comas.Tete.Cam_Axe_Horizontal[3].SegmentType := 1, [34].Comas.Tete.Cam_Axe_Horizontal[4].Master := 56.0, [34].Comas.Tete.Cam_Axe_Horizontal[4].Slave := 51.0, [34].Comas.Tete.Cam_Axe_Horizontal[5].Master := 66.0, [34].Comas.Tete.Cam_Axe_Horizontal[5].Slave := 61.0, [34].Comas.Tete.Cam_Axe_Horizontal[5].SegmentType := 1, [34].Comas.Tete.Cam_Axe_Horizontal[6].Master := 76.0, [34].Comas.Tete.Cam_Axe_Horizontal[6].Slave := 51.0, [34].Comas.Tete.Cam_Axe_Horizontal[6].SegmentType := 1, [34].Comas.Tete.Cam_Axe_Horizontal[7].Master := 94.0, [34].Comas.Tete.Cam_Axe_Vertical[1].Master := 1.0, [34].Comas.Tete.Cam_Axe_Vertical[2].Master := 11.0, [34].Comas.Tete.Cam_Axe_Vertical[3].Master := 41.0, [34].Comas.Tete.Cam_Axe_Vertical[3].Slave := -10.0, [34].Comas.Tete.Cam_Axe_Vertical[3].SegmentType := 1, [34].Comas.Tete.Cam_Axe_Vertical[4].Master := 62.0, [34].Comas.Tete.Cam_Axe_Vertical[4].Slave := 8.0, [34].Comas.Tete.Cam_Axe_Vertical[5].Master := 75.0, [34].Comas.Tete.Cam_Axe_Vertical[5].Slave := 17.0, [34].Comas.Tete.Cam_Axe_Vertical[5].SegmentType := 1, [34].Comas.Tete.Cam_Axe_Vertical[6].Master := 91.0, [34].Comas.Tete.Cam_Axe_Vertical[7].Master := 94.0, [34].Comas.Tete.Longueur_Cam_Axe_H := 8, [34].Comas.Tete.Offset_Vertical_Gauche := 38.0, [34].Comas.Tete.Offset_Horizontal_Gauche := 94.0, [34].Comas.Tete.Cam_Axe_Horizontal_Pan.B.x := 1.0, [34].Comas.Tete.Cam_Axe_Horizontal_Pan.C.x := 10.0, [34].Comas.Tete.Cam_Axe_Horizontal_Pan.C.y := 10.0,
        [34].Comas.Tete.Cam_Axe_Horizontal_Pan.D.x := 30.0, [34].Comas.Tete.Cam_Axe_Horizontal_Pan.D.y := 30.0, [34].Comas.Tete.Cam_Axe_Horizontal_Pan.E.x := 15.0, [34].Comas.Tete.Cam_Axe_Horizontal_Pan.E.y := 16.0, [34].Comas.Tete.Cam_Axe_Horizontal_Pan.F.x := 10.0, [34].Comas.Tete.Cam_Axe_Horizontal_Pan.F.y := 10.0, [34].Comas.Tete.Cam_Axe_Horizontal_Pan.G.x := 10.0, [34].Comas.Tete.Cam_Axe_Horizontal_Pan.G.y := -10.0, [34].Comas.Tete.Cam_Axe_Vertical_Pan.K.y := -10.0, [34].Comas.Tete.Cam_Axe_Vertical_Pan.L.x := 6.0, [34].Comas.Tete.Cam_Axe_Vertical_Pan.L.y := 8.0, [34].Comas.Tete.Cam_Axe_Vertical_Pan.M.x := 9.0, [34].Comas.Tete.Cam_Axe_Vertical_Pan.M.y := 17.0, [34].Comas.Tete.Cam_Axe_Vertical_Pan.N.x := 15.0, [34].Comas.Tete.Offset_Vertical_Droit := 45.0, [34].Comas.Tete.Offset_Horizontal_Droit := 94.0, [34].Comas.Tete.Reserve_Real1 := -5.0, [34].Comas.Pompe.Start_Cam_Logique_Avance := 1.0, [34].Comas.Pompe.Stop_Cam_Logique_Avance := 14.0, [34].Comas.Pompe.Start_Cam_Logique_Recul := 41.0, [34].Comas.Pompe.Stop_Cam_Logique_Recul := 41.0, [34].Comas.Pompe.Consigne_Vitesse_Avance := 34.0, [34].Comas.Pompe.Consigne_Acc_Dec_Avance := 40.0, [34].Comas.Pompe.Consigne_Jerk_Avance := 100.0, [34].Comas.Pompe.Consigne_Acc_Dec_Recul := 40.0, [34].Comas.Pompe.Consigne_Jerk_Recul := 100.0, [34].Comas.Pompe.Points_Pan.O.x := -10.0, [34].Comas.Pompe.Points_Pan.Q.x := 13.0, [34].Comas.Pompe.Reserve_Bool1 := 1, [34].Comas.Rouleaux.Consigne_Vitesse := 8.0, [34].Comas.Rouleaux.Consigne_Acc_Dec := 40.0, [34].Comas.Rouleaux.Consigne_Jerk := 100.0, [34].Comas.Rouleaux.Reserve_Real1 := -10.0, [34].Comas.Coupe_Fil.Activation := 1, [34].Comas.Coupe_Fil.Start_Cam_Logique_Virtuelle := 16.0, [34].Comas.Coupe_Fil.Stop_Cam_Logique_Virtuelle := 26.0, [34].Comas.Coupe_Fil.Consigne_Vitesse_Virtuelle := 280.0, [34].Comas.Coupe_Fil.Consigne_Acc_Dec_Virtuelle := 1000.0, [34].Comas.Coupe_Fil.Consigne_Jerk_Virtuelle := 50.0, [34].Comas.Coupe_Fil.Cam_Axe[0].SegmentType := 1, [34].Comas.Coupe_Fil.Cam_Axe[1].Master := 180.0, [34].Comas.Coupe_Fil.Cam_Axe[1].Slave := 180.0, [34].Comas.Coupe_Fil.Cam_Axe[2].Master := 250.0, [34].Comas.Coupe_Fil.Cam_Axe[2].Slave := 250.0, [34].Comas.Coupe_Fil.Cam_Axe[2].SegmentType := 1, [34].Comas.Coupe_Fil.Cam_Axe[3].Master := 360.0, [34].Comas.Coupe_Fil.Cam_Axe[3].Slave := 360.0, [34].Comas.Coupe_Fil.Cam_Axe[3].SegmentType := 1, [34].Comas.Coupe_Fil.Cam_Axe[4].SegmentType := 1, [34].Comas.Coupe_Fil.Points_Pan.W.x := -40.0, [34].Comas.Coupe_Fil.Reserve_Bool1 := 1, [34].Comas.Consigne_Vitesse_Manu_mm := 2.0, [34].Comas.Consigne_Acc_Decc_Manu_mm := 10.0, [34].Comas.Consigne_Jerk_Manu := 100.0, [34].Comas.Activation_Cam_Auto := 1, [34].Comas.Distance_CPT_Presence_Produit := 520, [34].Comas.Consigne_Vitesse_Manu_Tour := 10.0, [34].Comas.Consigne_Acc_Decc_Manu_Tour := 10.0, [34].Comas.Mode_Decoreuse_Cam_Logique := 1, [34].Comas.Reserve_Real6 := 200.0,
        [35].Name := 'palets breton MDLZ', [35].Comas.Pas_Machine := 74, [35].Comas.Came_Maitre[1].Master := 74.0, [35].Comas.Came_Maitre[1].Slave := 74.0, [35].Comas.Longueur_Came_Maitre := 2, [35].Comas.Tete.Stop_Cam_Logique_Degagement := 10.0, [35].Comas.Tete.Position_Degagement_H := 50.0, [35].Comas.Tete.Position_Degagement_V := 37.0, [35].Comas.Tete.Hauteur_Tete := -5, [35].Comas.Tete.Cam_Axe_Horizontal[1].Master := 3.0, [35].Comas.Tete.Cam_Axe_Horizontal[1].Slave := 1.0, [35].Comas.Tete.Cam_Axe_Horizontal[1].SegmentType := 1, [35].Comas.Tete.Cam_Axe_Horizontal[2].Master := 12.0, [35].Comas.Tete.Cam_Axe_Horizontal[2].Slave := 13.0, [35].Comas.Tete.Cam_Axe_Horizontal[3].Master := 28.0, [35].Comas.Tete.Cam_Axe_Horizontal[3].Slave := 20.0, [35].Comas.Tete.Cam_Axe_Horizontal[3].SegmentType := 1, [35].Comas.Tete.Cam_Axe_Horizontal[4].Master := 43.0, [35].Comas.Tete.Cam_Axe_Horizontal[4].Slave := 32.0, [35].Comas.Tete.Cam_Axe_Horizontal[5].Master := 53.0, [35].Comas.Tete.Cam_Axe_Horizontal[5].Slave := 22.0, [35].Comas.Tete.Cam_Axe_Horizontal[5].SegmentType := 1, [35].Comas.Tete.Cam_Axe_Horizontal[6].Master := 63.0, [35].Comas.Tete.Cam_Axe_Horizontal[6].Slave := 12.0, [35].Comas.Tete.Cam_Axe_Horizontal[6].SegmentType := 1, [35].Comas.Tete.Cam_Axe_Horizontal[7].Master := 74.0, [35].Comas.Tete.Cam_Axe_Vertical[1].Master := 3.0, [35].Comas.Tete.Cam_Axe_Vertical[2].Master := 12.0, [35].Comas.Tete.Cam_Axe_Vertical[3].Master := 28.0, [35].Comas.Tete.Cam_Axe_Vertical[3].Slave := -10.0, [35].Comas.Tete.Cam_Axe_Vertical[3].SegmentType := 1, [35].Comas.Tete.Cam_Axe_Vertical[4].Master := 49.0, [35].Comas.Tete.Cam_Axe_Vertical[4].Slave := 12.0, [35].Comas.Tete.Cam_Axe_Vertical[5].Master := 62.0, [35].Comas.Tete.Cam_Axe_Vertical[5].Slave := 17.0, [35].Comas.Tete.Cam_Axe_Vertical[5].SegmentType := 1, [35].Comas.Tete.Cam_Axe_Vertical[6].Master := 73.0, [35].Comas.Tete.Cam_Axe_Vertical[7].Master := 74.0, [35].Comas.Tete.Longueur_Cam_Axe_H := 8, [35].Comas.Tete.Offset_Vertical_Gauche := 38.0, [35].Comas.Tete.Offset_Horizontal_Gauche := 94.0, [35].Comas.Tete.Cam_Axe_Horizontal_Pan.B.x := 3.0, [35].Comas.Tete.Cam_Axe_Horizontal_Pan.B.y := 1.0, [35].Comas.Tete.Cam_Axe_Horizontal_Pan.C.x := 9.0, [35].Comas.Tete.Cam_Axe_Horizontal_Pan.C.y := 12.0, [35].Comas.Tete.Cam_Axe_Horizontal_Pan.D.x := 16.0, [35].Comas.Tete.Cam_Axe_Horizontal_Pan.D.y := 12.0, [35].Comas.Tete.Cam_Axe_Horizontal_Pan.E.x := 15.0, [35].Comas.Tete.Cam_Axe_Horizontal_Pan.E.y := 12.0, [35].Comas.Tete.Cam_Axe_Horizontal_Pan.F.x := 10.0, [35].Comas.Tete.Cam_Axe_Horizontal_Pan.F.y := -10.0, [35].Comas.Tete.Cam_Axe_Horizontal_Pan.G.x := 10.0, [35].Comas.Tete.Cam_Axe_Horizontal_Pan.G.y := -10.0, [35].Comas.Tete.Cam_Axe_Vertical_Pan.K.y := -10.0, [35].Comas.Tete.Cam_Axe_Vertical_Pan.L.x := 6.0, [35].Comas.Tete.Cam_Axe_Vertical_Pan.L.y := 12.0, [35].Comas.Tete.Cam_Axe_Vertical_Pan.M.x := 9.0, [35].Comas.Tete.Cam_Axe_Vertical_Pan.M.y := 17.0, [35].Comas.Tete.Cam_Axe_Vertical_Pan.N.x := 10.0, [35].Comas.Tete.Offset_Vertical_Droit := 45.0,
        [35].Comas.Tete.Offset_Horizontal_Droit := 94.0, [35].Comas.Tete.Reserve_Real1 := -5.0, [35].Comas.Pompe.Start_Cam_Logique_Avance := 2.0, [35].Comas.Pompe.Stop_Cam_Logique_Avance := 15.0, [35].Comas.Pompe.Start_Cam_Logique_Recul := 28.0, [35].Comas.Pompe.Stop_Cam_Logique_Recul := 28.0, [35].Comas.Pompe.Consigne_Vitesse_Avance := 40.0, [35].Comas.Pompe.Consigne_Acc_Dec_Avance := 40.0, [35].Comas.Pompe.Consigne_Jerk_Avance := 100.0, [35].Comas.Pompe.Consigne_Acc_Dec_Recul := 40.0, [35].Comas.Pompe.Consigne_Jerk_Recul := 100.0, [35].Comas.Pompe.Points_Pan.O.x := -10.0, [35].Comas.Pompe.Points_Pan.Q.x := 13.0, [35].Comas.Pompe.Reserve_Bool1 := 1, [35].Comas.Rouleaux.Consigne_Vitesse := 8.0, [35].Comas.Rouleaux.Consigne_Acc_Dec := 40.0, [35].Comas.Rouleaux.Consigne_Jerk := 100.0, [35].Comas.Rouleaux.Reserve_Real1 := -10.0, [35].Comas.Coupe_Fil.Activation := 1, [35].Comas.Coupe_Fil.Start_Cam_Logique_Virtuelle := 3.0, [35].Comas.Coupe_Fil.Stop_Cam_Logique_Virtuelle := 13.0, [35].Comas.Coupe_Fil.Consigne_Vitesse_Virtuelle := 290.0, [35].Comas.Coupe_Fil.Consigne_Acc_Dec_Virtuelle := 1000.0, [35].Comas.Coupe_Fil.Consigne_Jerk_Virtuelle := 50.0, [35].Comas.Coupe_Fil.Cam_Axe[0].SegmentType := 1, [35].Comas.Coupe_Fil.Cam_Axe[1].Master := 180.0, [35].Comas.Coupe_Fil.Cam_Axe[1].Slave := 180.0, [35].Comas.Coupe_Fil.Cam_Axe[2].Master := 250.0, [35].Comas.Coupe_Fil.Cam_Axe[2].Slave := 350.0, [35].Comas.Coupe_Fil.Cam_Axe[2].SegmentType := 1, [35].Comas.Coupe_Fil.Cam_Axe[3].Master := 360.0, [35].Comas.Coupe_Fil.Cam_Axe[3].Slave := 360.0, [35].Comas.Coupe_Fil.Cam_Axe[3].SegmentType := 1, [35].Comas.Coupe_Fil.Cam_Axe[4].SegmentType := 1, [35].Comas.Coupe_Fil.Points_Pan.W.x := -40.0, [35].Comas.Coupe_Fil.Reserve_Bool1 := 1, [35].Comas.Consigne_Vitesse_Manu_mm := 2.0, [35].Comas.Consigne_Acc_Decc_Manu_mm := 10.0, [35].Comas.Consigne_Jerk_Manu := 100.0, [35].Comas.Activation_Cam_Auto := 1, [35].Comas.Distance_CPT_Presence_Produit := 520, [35].Comas.Consigne_Vitesse_Manu_Tour := 10.0, [35].Comas.Consigne_Acc_Decc_Manu_Tour := 10.0, [35].Comas.Mode_Decoreuse_Cam_Logique := 1, [35].Comas.Reserve_Real3 := 1.0, [35].Comas.Reserve_Real4 := 1.0, [35].Comas.Reserve_Real5 := 5.0, [35].Comas.Reserve_Real6 := 200.0, [35].Reserve_Real2 := 200.0, [35].Reserve_Real3 := 10.0, [36].Name := 'galettes d$'avoine', [36].Comas.Pas_Machine := 78, [36].Comas.Came_Maitre[1].Master := 78.0, [36].Comas.Came_Maitre[1].Slave := 78.0, [36].Comas.Longueur_Came_Maitre := 2, [36].Comas.Tete.Stop_Cam_Logique_Degagement := 10.0, [36].Comas.Tete.Position_Degagement_H := 50.0, [36].Comas.Tete.Position_Degagement_V := 37.0, [36].Comas.Tete.Hauteur_Tete := -20, [36].Comas.Tete.Cam_Axe_Horizontal[1].Master := 1.0,
        [36].Comas.Tete.Cam_Axe_Horizontal[2].Master := 11.0, [36].Comas.Tete.Cam_Axe_Horizontal[2].Slave := -3.0, [36].Comas.Tete.Cam_Axe_Horizontal[3].Master := 41.0, [36].Comas.Tete.Cam_Axe_Horizontal[3].Slave := -6.0, [36].Comas.Tete.Cam_Axe_Horizontal[3].SegmentType := 1, [36].Comas.Tete.Cam_Axe_Horizontal[4].Master := 53.0, [36].Comas.Tete.Cam_Axe_Horizontal[4].Slave := 4.0, [36].Comas.Tete.Cam_Axe_Horizontal[4].SegmentType := 1, [36].Comas.Tete.Cam_Axe_Horizontal[5].Master := 63.0, [36].Comas.Tete.Cam_Axe_Horizontal[5].Slave := 9.0, [36].Comas.Tete.Cam_Axe_Horizontal[5].SegmentType := 1, [36].Comas.Tete.Cam_Axe_Horizontal[6].Master := 73.0, [36].Comas.Tete.Cam_Axe_Horizontal[6].Slave := 4.0, [36].Comas.Tete.Cam_Axe_Horizontal[6].SegmentType := 1, [36].Comas.Tete.Cam_Axe_Horizontal[7].Master := 78.0, [36].Comas.Tete.Cam_Axe_Vertical[1].Master := 1.0, [36].Comas.Tete.Cam_Axe_Vertical[2].Master := 11.0, [36].Comas.Tete.Cam_Axe_Vertical[3].Master := 41.0, [36].Comas.Tete.Cam_Axe_Vertical[3].SegmentType := 1, [36].Comas.Tete.Cam_Axe_Vertical[4].Master := 53.0, [36].Comas.Tete.Cam_Axe_Vertical[4].Slave := 15.0, [36].Comas.Tete.Cam_Axe_Vertical[5].Master := 63.0, [36].Comas.Tete.Cam_Axe_Vertical[5].Slave := 20.0, [36].Comas.Tete.Cam_Axe_Vertical[5].SegmentType := 1, [36].Comas.Tete.Cam_Axe_Vertical[6].Master := 73.0, [36].Comas.Tete.Cam_Axe_Vertical[6].Slave := 12.0, [36].Comas.Tete.Cam_Axe_Vertical[6].SegmentType := 1, [36].Comas.Tete.Cam_Axe_Vertical[7].Master := 78.0, [36].Comas.Tete.Longueur_Cam_Axe_H := 8, [36].Comas.Tete.Offset_Vertical_Gauche := 38.0, [36].Comas.Tete.Offset_Horizontal_Gauche := 94.0, [36].Comas.Tete.Cam_Axe_Horizontal_Pan.B.x := 1.0, [36].Comas.Tete.Cam_Axe_Horizontal_Pan.C.x := 10.0, [36].Comas.Tete.Cam_Axe_Horizontal_Pan.C.y := -3.0, [36].Comas.Tete.Cam_Axe_Horizontal_Pan.D.x := 30.0, [36].Comas.Tete.Cam_Axe_Horizontal_Pan.D.y := 5.0, [36].Comas.Tete.Cam_Axe_Horizontal_Pan.E.x := 12.0, [36].Comas.Tete.Cam_Axe_Horizontal_Pan.E.y := 10.0, [36].Comas.Tete.Cam_Axe_Horizontal_Pan.F.x := 10.0, [36].Comas.Tete.Cam_Axe_Horizontal_Pan.F.y := 5.0, [36].Comas.Tete.Cam_Axe_Horizontal_Pan.G.x := 10.0, [36].Comas.Tete.Cam_Axe_Horizontal_Pan.G.y := -5.0, [36].Comas.Tete.Cam_Axe_Vertical_Pan.L.y := 15.0, [36].Comas.Tete.Cam_Axe_Vertical_Pan.M.y := 20.0, [36].Comas.Tete.Cam_Axe_Vertical_Pan.N.y := 12.0, [36].Comas.Tete.Offset_Vertical_Droit := 45.0, [36].Comas.Tete.Offset_Horizontal_Droit := 94.0, [36].Comas.Tete.Reserve_Real1 := -8.0, [36].Comas.Pompe.Start_Cam_Logique_Avance := 1.0, [36].Comas.Pompe.Stop_Cam_Logique_Avance := 14.0, [36].Comas.Pompe.Start_Cam_Logique_Recul := 41.0, [36].Comas.Pompe.Stop_Cam_Logique_Recul := 41.0, [36].Comas.Pompe.Consigne_Vitesse_Avance := 19.6, [36].Comas.Pompe.Consigne_Acc_Dec_Avance := 40.0, [36].Comas.Pompe.Consigne_Jerk_Avance := 100.0, [36].Comas.Pompe.Consigne_Acc_Dec_Recul := 40.0, [36].Comas.Pompe.Consigne_Jerk_Recul := 100.0, [36].Comas.Pompe.Points_Pan.O.x := -10.0, [36].Comas.Pompe.Points_Pan.Q.x := 13.0, [36].Comas.Pompe.Reserve_Bool1 := 1,
        [36].Comas.Rouleaux.Consigne_Vitesse := 18.5, [36].Comas.Rouleaux.Consigne_Acc_Dec := 40.0, [36].Comas.Rouleaux.Consigne_Jerk := 100.0, [36].Comas.Rouleaux.Reserve_Real1 := -10.0, [36].Comas.Coupe_Fil.Activation := 1, [36].Comas.Coupe_Fil.Start_Cam_Logique_Virtuelle := 18.0, [36].Comas.Coupe_Fil.Stop_Cam_Logique_Virtuelle := 28.0, [36].Comas.Coupe_Fil.Consigne_Vitesse_Virtuelle := 400.0, [36].Comas.Coupe_Fil.Consigne_Acc_Dec_Virtuelle := 1200.0, [36].Comas.Coupe_Fil.Consigne_Jerk_Virtuelle := 50.0, [36].Comas.Coupe_Fil.Cam_Axe[0].SegmentType := 1, [36].Comas.Coupe_Fil.Cam_Axe[1].Master := 180.0, [36].Comas.Coupe_Fil.Cam_Axe[1].Slave := 180.0, [36].Comas.Coupe_Fil.Cam_Axe[2].Master := 250.0, [36].Comas.Coupe_Fil.Cam_Axe[2].Slave := 200.0, [36].Comas.Coupe_Fil.Cam_Axe[2].SegmentType := 1, [36].Comas.Coupe_Fil.Cam_Axe[3].Master := 360.0, [36].Comas.Coupe_Fil.Cam_Axe[3].Slave := 360.0, [36].Comas.Coupe_Fil.Cam_Axe[3].SegmentType := 1, [36].Comas.Coupe_Fil.Cam_Axe[4].SegmentType := 1, [36].Comas.Coupe_Fil.Points_Pan.W.x := -35.0, [36].Comas.Coupe_Fil.Reserve_Bool1 := 1, [36].Comas.Consigne_Vitesse_Manu_mm := 2.0, [36].Comas.Consigne_Acc_Decc_Manu_mm := 10.0, [36].Comas.Consigne_Jerk_Manu := 100.0, [36].Comas.Activation_Cam_Auto := 1, [36].Comas.Distance_CPT_Presence_Produit := 520, [36].Comas.Consigne_Vitesse_Manu_Tour := 10.0, [36].Comas.Consigne_Acc_Decc_Manu_Tour := 10.0, [36].Comas.Mode_Decoreuse_Cam_Logique := 1, [36].Comas.Reserve_Real3 := 1.0, [36].Comas.Reserve_Real4 := 1.0, [36].Comas.Reserve_Real5 := 5.0, [36].Comas.Reserve_Real6 := 200.0, [36].Reserve_Real2 := 200.0, [36].Reserve_Real3 := 10.0, [37].Comas.Reserve_Real6 := 200.0, [38].Comas.Reserve_Real6 := 200.0, [39].Comas.Reserve_Real6 := 200.0, [40].Name := 'test linea', [40].Comas.Pas_Machine := 80, [40].Comas.Came_Maitre[1].Master := 80.0, [40].Comas.Came_Maitre[1].Slave := 80.0, [40].Comas.Longueur_Came_Maitre := 2, [40].Comas.Tete.Stop_Cam_Logique_Degagement := 10.0, [40].Comas.Tete.Position_Degagement_H := 50.0, [40].Comas.Tete.Position_Degagement_V := 35.0, [40].Comas.Tete.Hauteur_Tete := -10, [40].Comas.Tete.Cam_Axe_Horizontal[1].Master := 1.0, [40].Comas.Tete.Cam_Axe_Horizontal[2].Master := 7.0, [40].Comas.Tete.Cam_Axe_Horizontal[2].Slave := 2.0, [40].Comas.Tete.Cam_Axe_Horizontal[3].Master := 25.0, [40].Comas.Tete.Cam_Axe_Horizontal[3].Slave := 26.5, [40].Comas.Tete.Cam_Axe_Horizontal[3].SegmentType := 1, [40].Comas.Tete.Cam_Axe_Horizontal[4].Master := 35.0, [40].Comas.Tete.Cam_Axe_Horizontal[4].Slave := 46.5, [40].Comas.Tete.Cam_Axe_Horizontal[5].Master := 40.0, [40].Comas.Tete.Cam_Axe_Horizontal[5].Slave := 46.5, [40].Comas.Tete.Cam_Axe_Horizontal[6].Master := 50.0, [40].Comas.Tete.Cam_Axe_Horizontal[6].Slave := 46.5,
        [40].Comas.Tete.Cam_Axe_Horizontal[6].SegmentType := 1, [40].Comas.Tete.Cam_Axe_Horizontal[7].Master := 80.0, [40].Comas.Tete.Cam_Axe_Vertical[0].Slave := 15.0, [40].Comas.Tete.Cam_Axe_Vertical[1].Master := 1.0, [40].Comas.Tete.Cam_Axe_Vertical[1].Slave := 15.0, [40].Comas.Tete.Cam_Axe_Vertical[2].Master := 10.0, [40].Comas.Tete.Cam_Axe_Vertical[2].Slave := 15.0, [40].Comas.Tete.Cam_Axe_Vertical[3].Master := 30.0, [40].Comas.Tete.Cam_Axe_Vertical[3].Slave := 15.0, [40].Comas.Tete.Cam_Axe_Vertical[3].SegmentType := 1, [40].Comas.Tete.Cam_Axe_Vertical[4].Master := 40.0, [40].Comas.Tete.Cam_Axe_Vertical[4].Slave := 40.0, [40].Comas.Tete.Cam_Axe_Vertical[5].Master := 45.0, [40].Comas.Tete.Cam_Axe_Vertical[5].Slave := 30.0, [40].Comas.Tete.Cam_Axe_Vertical[5].SegmentType := 1, [40].Comas.Tete.Cam_Axe_Vertical[6].Master := 54.0, [40].Comas.Tete.Cam_Axe_Vertical[6].Slave := 15.0, [40].Comas.Tete.Cam_Axe_Vertical[7].Master := 80.0, [40].Comas.Tete.Cam_Axe_Vertical[7].Slave := 15.0, [40].Comas.Tete.Longueur_Cam_Axe_H := 8, [40].Comas.Tete.Offset_Vertical_Gauche := 38.0, [40].Comas.Tete.Offset_Horizontal_Gauche := 95.0, [40].Comas.Tete.Cam_Axe_Horizontal_Pan.B.x := 1.0, [40].Comas.Tete.Cam_Axe_Horizontal_Pan.C.x := 6.0, [40].Comas.Tete.Cam_Axe_Horizontal_Pan.C.y := 2.0, [40].Comas.Tete.Cam_Axe_Horizontal_Pan.D.x := 18.0, [40].Comas.Tete.Cam_Axe_Horizontal_Pan.D.y := 20.0, [40].Comas.Tete.Cam_Axe_Horizontal_Pan.E.x := 10.0, [40].Comas.Tete.Cam_Axe_Horizontal_Pan.E.y := 20.0, [40].Comas.Tete.Cam_Axe_Horizontal_Pan.F.x := 5.0, [40].Comas.Tete.Cam_Axe_Horizontal_Pan.G.x := 10.0, [40].Comas.Tete.Cam_Axe_Vertical_Pan.H.y := 15.0, [40].Comas.Tete.Cam_Axe_Vertical_Pan.I.y := 15.0, [40].Comas.Tete.Cam_Axe_Vertical_Pan.J.x := 3.0, [40].Comas.Tete.Cam_Axe_Vertical_Pan.J.y := 15.0, [40].Comas.Tete.Cam_Axe_Vertical_Pan.K.x := 5.0, [40].Comas.Tete.Cam_Axe_Vertical_Pan.K.y := 15.0, [40].Comas.Tete.Cam_Axe_Vertical_Pan.L.x := 5.0, [40].Comas.Tete.Cam_Axe_Vertical_Pan.L.y := 40.0, [40].Comas.Tete.Cam_Axe_Vertical_Pan.M.x := 5.0, [40].Comas.Tete.Cam_Axe_Vertical_Pan.M.y := 30.0, [40].Comas.Tete.Cam_Axe_Vertical_Pan.N.x := 4.0, [40].Comas.Tete.Cam_Axe_Vertical_Pan.N.y := 15.0, [40].Comas.Tete.Offset_Vertical_Droit := 45.0, [40].Comas.Tete.Offset_Horizontal_Droit := 95.0, [40].Comas.Tete.Reserve_Real1 := 4.5, [40].Comas.Pompe.Start_Cam_Logique_Avance := -15.0, [40].Comas.Pompe.Stop_Cam_Logique_Avance := 10.0, [40].Comas.Pompe.Start_Cam_Logique_Recul := 30.0, [40].Comas.Pompe.Stop_Cam_Logique_Recul := 30.0, [40].Comas.Pompe.Consigne_Vitesse_Avance := 10.0, [40].Comas.Pompe.Consigne_Acc_Dec_Avance := 40.0, [40].Comas.Pompe.Consigne_Jerk_Avance := 100.0, [40].Comas.Pompe.Consigne_Vitesse_Recul := -14.0, [40].Comas.Pompe.Consigne_Acc_Dec_Recul := 40.0, [40].Comas.Pompe.Consigne_Jerk_Recul := 100.0, [40].Comas.Pompe.Points_Pan.O.x := -40.0, [40].Comas.Pompe.Start_Cam_Logique_Inter1 := 10.0, [40].Comas.Pompe.Stop_Cam_Logique_Inter1 := 13.0, [40].Comas.Pompe.Consigne_Vitesse_Inter1 := -9.0,
        [40].Comas.Rouleaux.Syncho_Pompe := 1, [40].Comas.Rouleaux.Consigne_Vitesse := 25.0, [40].Comas.Rouleaux.Consigne_Acc_Dec := 40.0, [40].Comas.Rouleaux.Consigne_Jerk := 100.0, [40].Comas.Coupe_Fil.Start_Cam_Logique_Virtuelle := 11.0, [40].Comas.Coupe_Fil.Stop_Cam_Logique_Virtuelle := 21.0, [40].Comas.Coupe_Fil.Consigne_Vitesse_Virtuelle := 200.0, [40].Comas.Coupe_Fil.Consigne_Acc_Dec_Virtuelle := 1000.0, [40].Comas.Coupe_Fil.Consigne_Jerk_Virtuelle := 50.0, [40].Comas.Coupe_Fil.Cam_Axe[0].SegmentType := 1, [40].Comas.Coupe_Fil.Cam_Axe[1].Master := 180.0, [40].Comas.Coupe_Fil.Cam_Axe[1].Slave := 90.0, [40].Comas.Coupe_Fil.Cam_Axe[2].Master := 360.0, [40].Comas.Coupe_Fil.Cam_Axe[2].Slave := 360.0, [40].Comas.Coupe_Fil.Cam_Axe[2].SegmentType := 1, [40].Comas.Coupe_Fil.Points_Pan.W.x := 30.0, [40].Comas.Consigne_Vitesse_Manu_mm := 2.0, [40].Comas.Consigne_Acc_Decc_Manu_mm := 10.0, [40].Comas.Consigne_Jerk_Manu := 100.0, [40].Comas.Activation_Cam_Auto := 1, [40].Comas.Mode_CPT_Presence := 1, [40].Comas.Distance_CPT_Presence_Produit := 513, [40].Comas.Consigne_Vitesse_Manu_Tour := 10.0, [40].Comas.Consigne_Acc_Decc_Manu_Tour := 10.0, [40].Comas.Mode_Decoreuse_Cam_Logique := 1, [40].Comas.Reserve_Real3 := 1.0, [40].Comas.Reserve_Real4 := 1.0, [40].Comas.Reserve_Real5 := 30.0, [40].Comas.Reserve_Bool1 := 1, [40].Comas.Reserve_Real6 := 200.0, [41].Name := 'tes coupe fil inverse', [41].Comas.Pas_Machine := 100, [41].Comas.Came_Maitre[1].Master := 100.0, [41].Comas.Came_Maitre[1].Slave := 100.0, [41].Comas.Longueur_Came_Maitre := 2, [41].Comas.Tete.Stop_Cam_Logique_Degagement := 10.0, [41].Comas.Tete.Position_Degagement_H := 50.0, [41].Comas.Tete.Position_Degagement_V := 35.0, [41].Comas.Tete.Hauteur_Tete := 10, [41].Comas.Tete.Cam_Axe_Horizontal[1].Master := 1.0, [41].Comas.Tete.Cam_Axe_Horizontal[1].SegmentType := 1, [41].Comas.Tete.Cam_Axe_Horizontal[2].Master := 11.0, [41].Comas.Tete.Cam_Axe_Horizontal[3].Master := 16.0, [41].Comas.Tete.Cam_Axe_Horizontal[3].SegmentType := 1, [41].Comas.Tete.Cam_Axe_Horizontal[4].Master := 26.0, [41].Comas.Tete.Cam_Axe_Horizontal[4].Slave := 5.0, [41].Comas.Tete.Cam_Axe_Horizontal[4].SegmentType := 1, [41].Comas.Tete.Cam_Axe_Horizontal[5].Master := 36.0, [41].Comas.Tete.Cam_Axe_Horizontal[5].Slave := 5.0, [41].Comas.Tete.Cam_Axe_Horizontal[5].SegmentType := 1, [41].Comas.Tete.Cam_Axe_Horizontal[6].Master := 46.0, [41].Comas.Tete.Cam_Axe_Horizontal[6].SegmentType := 1, [41].Comas.Tete.Cam_Axe_Horizontal[7].Master := 100.0, [41].Comas.Tete.Cam_Axe_Vertical[1].Master := 1.0, [41].Comas.Tete.Cam_Axe_Vertical[2].Master := 11.0, [41].Comas.Tete.Cam_Axe_Vertical[3].Master := 16.0, [41].Comas.Tete.Cam_Axe_Vertical[3].SegmentType := 1, [41].Comas.Tete.Cam_Axe_Vertical[4].Master := 31.0, [41].Comas.Tete.Cam_Axe_Vertical[5].Master := 51.0, [41].Comas.Tete.Cam_Axe_Vertical[5].SegmentType := 1,
        [41].Comas.Tete.Cam_Axe_Vertical[6].Master := 61.0, [41].Comas.Tete.Cam_Axe_Vertical[7].Master := 100.0, [41].Comas.Tete.Longueur_Cam_Axe_H := 8, [41].Comas.Tete.Offset_Vertical_Gauche := 38.0, [41].Comas.Tete.Offset_Horizontal_Gauche := 95.0, [41].Comas.Tete.Cam_Axe_Horizontal_Pan.B.x := 1.0, [41].Comas.Tete.Cam_Axe_Horizontal_Pan.C.x := 10.0, [41].Comas.Tete.Cam_Axe_Horizontal_Pan.D.x := 5.0, [41].Comas.Tete.Cam_Axe_Horizontal_Pan.E.x := 10.0, [41].Comas.Tete.Cam_Axe_Horizontal_Pan.E.y := 5.0, [41].Comas.Tete.Cam_Axe_Horizontal_Pan.F.x := 10.0, [41].Comas.Tete.Cam_Axe_Horizontal_Pan.G.x := 10.0, [41].Comas.Tete.Cam_Axe_Horizontal_Pan.G.y := -5.0, [41].Comas.Tete.Cam_Axe_Vertical_Pan.L.x := 5.0, [41].Comas.Tete.Cam_Axe_Vertical_Pan.M.x := 15.0, [41].Comas.Tete.Cam_Axe_Vertical_Pan.N.x := 15.0, [41].Comas.Tete.Offset_Vertical_Droit := 45.0, [41].Comas.Tete.Offset_Horizontal_Droit := 95.0, [41].Comas.Pompe.Start_Cam_Logique_Avance := -32.0, [41].Comas.Pompe.Stop_Cam_Logique_Avance := -1.0, [41].Comas.Pompe.Start_Cam_Logique_Recul := -9.0, [41].Comas.Pompe.Stop_Cam_Logique_Recul := 6.0, [41].Comas.Pompe.Consigne_Vitesse_Avance := 19.0, [41].Comas.Pompe.Consigne_Acc_Dec_Avance := 40.0, [41].Comas.Pompe.Consigne_Jerk_Avance := 100.0, [41].Comas.Pompe.Consigne_Acc_Dec_Recul := 40.0, [41].Comas.Pompe.Consigne_Jerk_Recul := 100.0, [41].Comas.Pompe.Points_Pan.O.x := -43.0, [41].Comas.Pompe.Points_Pan.Q.x := 31.0, [41].Comas.Pompe.Points_Pan.S.x := -25.0, [41].Comas.Pompe.Points_Pan.U.x := 15.0, [41].Comas.Pompe.Reserve_Bool1 := 1, [41].Comas.Rouleaux.Syncho_Pompe := 1, [41].Comas.Rouleaux.Consigne_Vitesse := 30.0, [41].Comas.Rouleaux.Consigne_Acc_Dec := 40.0, [41].Comas.Rouleaux.Consigne_Jerk := 100.0, [41].Comas.Coupe_Fil.Activation := 1, [41].Comas.Coupe_Fil.Start_Cam_Logique_Virtuelle := 12.5, [41].Comas.Coupe_Fil.Stop_Cam_Logique_Virtuelle := 22.5, [41].Comas.Coupe_Fil.Consigne_Vitesse_Virtuelle := 250.0, [41].Comas.Coupe_Fil.Consigne_Acc_Dec_Virtuelle := 850.0, [41].Comas.Coupe_Fil.Consigne_Jerk_Virtuelle := 50.0, [41].Comas.Coupe_Fil.Cam_Axe[0].SegmentType := 1, [41].Comas.Coupe_Fil.Cam_Axe[1].Master := 180.0, [41].Comas.Coupe_Fil.Cam_Axe[1].Slave := -180.0, [41].Comas.Coupe_Fil.Cam_Axe[2].Master := 250.0, [41].Comas.Coupe_Fil.Cam_Axe[2].Slave := -200.0, [41].Comas.Coupe_Fil.Cam_Axe[3].Master := 300.0, [41].Comas.Coupe_Fil.Cam_Axe[3].Slave := -210.0, [41].Comas.Coupe_Fil.Cam_Axe[3].SegmentType := 1, [41].Comas.Coupe_Fil.Cam_Axe[4].Master := 360.0, [41].Comas.Coupe_Fil.Cam_Axe[4].Slave := -360.0, [41].Comas.Coupe_Fil.Cam_Axe[4].SegmentType := 1, [41].Comas.Coupe_Fil.Points_Pan.W.x := -13.5, [41].Comas.Coupe_Fil.Reserve_Bool1 := 1, [41].Comas.Consigne_Vitesse_Manu_mm := 2.0, [41].Comas.Consigne_Acc_Decc_Manu_mm := 10.0, [41].Comas.Consigne_Jerk_Manu := 100.0, [41].Comas.Activation_Cam_Auto := 1, [41].Comas.Distance_CPT_Presence_Produit := 520,
        [41].Comas.Consigne_Vitesse_Manu_Tour := 10.0, [41].Comas.Consigne_Acc_Decc_Manu_Tour := 10.0, [41].Comas.Mode_Decoreuse_Cam_Logique := 1, [41].Comas.Reserve_Real3 := 1.0, [41].Comas.Reserve_Real4 := 1.0, [41].Comas.Reserve_Real5 := 5.0, [41].Comas.Reserve_Real6 := 5.0, [42].Name := 'test buse rotative', [42].Comas.Pas_Machine := 40, [42].Comas.Came_Maitre[1].Master := 40.0, [42].Comas.Came_Maitre[1].Slave := 40.0, [42].Comas.Longueur_Came_Maitre := 2, [42].Comas.Tete.Stop_Cam_Logique_Degagement := 10.0, [42].Comas.Tete.Position_Degagement_H := 50.0, [42].Comas.Tete.Position_Degagement_V := 37.0, [42].Comas.Tete.Hauteur_Tete := -7, [42].Comas.Tete.Cam_Axe_Horizontal[2].Slave := -3.0, [42].Comas.Tete.Cam_Axe_Horizontal[3].Slave := -3.0, [42].Comas.Tete.Cam_Axe_Horizontal[3].SegmentType := 1, [42].Comas.Tete.Cam_Axe_Horizontal[4].Slave := 7.0, [42].Comas.Tete.Cam_Axe_Horizontal[4].SegmentType := 1, [42].Comas.Tete.Cam_Axe_Horizontal[5].Slave := 12.0, [42].Comas.Tete.Cam_Axe_Horizontal[5].SegmentType := 1, [42].Comas.Tete.Cam_Axe_Horizontal[6].Slave := 2.0, [42].Comas.Tete.Cam_Axe_Horizontal[6].SegmentType := 1, [42].Comas.Tete.Cam_Axe_Horizontal[7].Master := 40.0, [42].Comas.Tete.Cam_Axe_Vertical[3].SegmentType := 1, [42].Comas.Tete.Cam_Axe_Vertical[4].Slave := 12.0, [42].Comas.Tete.Cam_Axe_Vertical[5].Slave := 18.0, [42].Comas.Tete.Cam_Axe_Vertical[5].SegmentType := 1, [42].Comas.Tete.Cam_Axe_Vertical[7].Master := 40.0, [42].Comas.Tete.Longueur_Cam_Axe_H := 8, [42].Comas.Tete.Offset_Vertical_Gauche := 38.0, [42].Comas.Tete.Offset_Horizontal_Gauche := 94.0, [42].Comas.Tete.Cam_Axe_Horizontal_Pan.C.y := -3.0, [42].Comas.Tete.Cam_Axe_Horizontal_Pan.D.y := 5.0, [42].Comas.Tete.Cam_Axe_Horizontal_Pan.E.y := 10.0, [42].Comas.Tete.Cam_Axe_Horizontal_Pan.F.y := 5.0, [42].Comas.Tete.Cam_Axe_Horizontal_Pan.G.y := -10.0, [42].Comas.Tete.Cam_Axe_Vertical_Pan.L.y := 12.0, [42].Comas.Tete.Cam_Axe_Vertical_Pan.M.y := 18.0, [42].Comas.Tete.Offset_Vertical_Droit := 45.0, [42].Comas.Tete.Offset_Horizontal_Droit := 94.0, [42].Comas.Tete.Reserve_Real1 := -5.0, [42].Comas.Pompe.Stop_Cam_Logique_Avance := 40.0, [42].Comas.Pompe.Consigne_Vitesse_Avance := 16.0, [42].Comas.Pompe.Consigne_Acc_Dec_Avance := 40.0, [42].Comas.Pompe.Consigne_Jerk_Avance := 100.0, [42].Comas.Pompe.Consigne_Acc_Dec_Recul := 40.0, [42].Comas.Pompe.Consigne_Jerk_Recul := 100.0, [42].Comas.Pompe.Points_Pan.Q.x := 40.0, [42].Comas.Pompe.Reserve_Bool1 := 1, [42].Comas.Rouleaux.Consigne_Vitesse := 30.0, [42].Comas.Rouleaux.Consigne_Acc_Dec := 40.0, [42].Comas.Rouleaux.Consigne_Jerk := 100.0, [42].Comas.Rouleaux.Reserve_Real1 := -10.0, [42].Comas.Coupe_Fil.Activation := 1, [42].Comas.Coupe_Fil.Start_Cam_Logique_Virtuelle := -35.0, [42].Comas.Coupe_Fil.Stop_Cam_Logique_Virtuelle := -25.0, [42].Comas.Coupe_Fil.Consigne_Vitesse_Virtuelle := 300.0,
        [42].Comas.Coupe_Fil.Consigne_Acc_Dec_Virtuelle := 300.0, [42].Comas.Coupe_Fil.Consigne_Jerk_Virtuelle := 50.0, [42].Comas.Coupe_Fil.Cam_Axe[1].Master := 90.0, [42].Comas.Coupe_Fil.Cam_Axe[1].Slave := 5.7, [42].Comas.Coupe_Fil.Cam_Axe[2].Master := 180.0, [42].Comas.Coupe_Fil.Cam_Axe[3].Master := 270.0, [42].Comas.Coupe_Fil.Cam_Axe[3].Slave := 5.7, [42].Comas.Coupe_Fil.Cam_Axe[4].Master := 360.0, [42].Comas.Coupe_Fil.Offset_Axe := 8.0, [42].Comas.Coupe_Fil.Points_Pan.W.x := -35.0, [42].Comas.Coupe_Fil.Reserve_Bool5 := 1, [42].Comas.Consigne_Vitesse_Manu_mm := 2.0, [42].Comas.Consigne_Acc_Decc_Manu_mm := 10.0, [42].Comas.Consigne_Jerk_Manu := 100.0, [42].Comas.Distance_CPT_Presence_Produit := 520, [42].Comas.Consigne_Vitesse_Manu_Tour := 10.0, [42].Comas.Consigne_Acc_Decc_Manu_Tour := 10.0, [42].Comas.Mode_Decoreuse_Cam_Logique := 1, [42].Comas.Reserve_Real3 := 1.0, [42].Comas.Reserve_Real4 := 1.0, [42].Comas.Reserve_Real5 := 5.0, [42].Comas.Reserve_Real6 := 197.0, [42].Reserve_Real2 := 200.0, [42].Reserve_Real3 := 10.0, [43].Comas.Reserve_Real6 := 200.0, [44].Comas.Reserve_Real6 := 200.0, [45].Comas.Reserve_Real6 := 200.0, [46].Comas.Reserve_Real6 := 200.0, [47].Comas.Reserve_Real6 := 200.0, [48].Comas.Reserve_Real6 := 200.0, [49].Comas.Reserve_Real6 := 200.0);
   Resynchro_Codeur : BOOL;
   Resynchro_Codeur_Front : BOOL;
   RSW_Acquit_defaut : BOOL;
   RSW_BADGE_Numero_Page : DINT;
   RSW_BADGE_Numero_Page_En_Cours : DINT := 99;
   RSW_BADGE_RAZ_CODE : BOOL;
   RSW_BADGE_Temps_Restant : DINT;
   RSW_BADGE_TOF_Chagement_Page : TIMER := (PRE := 2000, ACC := 2000);
   RSW_CO_Activation_Nettoyage : BOOL;
   RSW_CO_BP_Coupe_Fil_Neg : BOOL;
   RSW_CO_BP_Coupe_Fil_Pos : BOOL;
   RSW_CO_BP_Horizontal_Droit_Neg : BOOL;
   RSW_CO_BP_Horizontal_Droit_Pos : BOOL;
   RSW_CO_BP_Horizontal_Gauche_Neg : BOOL;
   RSW_CO_BP_Horizontal_Gauche_Pos : BOOL;
   RSW_CO_BP_Horizontal_Neg : BOOL;
   RSW_CO_BP_Horizontal_Pos : BOOL;
   RSW_CO_BP_Pompe_Doseuse_Neg : BOOL;
   RSW_CO_BP_Pompe_Doseuse_Pos : BOOL;
   RSW_CO_BP_Rouleaux_Canneles_Neg : BOOL;
   RSW_CO_BP_Rouleaux_Canneles_Pos : BOOL;
   RSW_CO_BP_Vertical_Droit_Neg : BOOL;
   RSW_CO_BP_Vertical_Droit_Pos : BOOL;
   RSW_CO_BP_Vertical_Gauche_Neg : BOOL;
   RSW_CO_BP_Vertical_Gauche_Pos : BOOL;
   RSW_CO_BP_Vertical_Neg : BOOL;
   RSW_CO_BP_Vertical_Pos : BOOL;
   RSW_CO_Commande_Unitaire : BOOL := 1;
   RSW_CO_Demande_Initialisation : BOOL;
   RSW_CO_NB_Rangs_minutes : REAL := 31.012836;
   RSW_Depose_Active : BOOL := 1;
   RSW_Niveau_Accu_LA : DINT := 40;
   RSW_Niveau_Accu_LD : DINT := 3;
   SOR_CO_Echange_Amont_OK : ALIAS FOR Local:3:O.Pt07.Data;
   SOR_CO_Top_Debut_Cycle_Decoreuse : ALIAS FOR Local:3:O.Pt05.Data;
   SOR_CO_Top_Debut_Dosage : ALIAS FOR Local:3:O.Pt06.Data;
   SOR_CO_Voyant_Arret : ALIAS FOR Local:3:O.Pt01.Data;
   SOR_CO_Voyant_Marche : ALIAS FOR Local:3:O.Pt00.Data;
   SOR_CO_Voyant_Rearmement : ALIAS FOR Local:3:O.Pt02.Data;
   Speed_Control_Pompe : Axis_speed_control := (Enable := 1, Acc := 40.0, Dec := 40.0, Jerk := 100.0);
   Speed_Control_Rouleaux : Axis_speed_control := (Enable := 1, Acc := 40.0, Dec := 40.0, Jerk := 100.0);
   Start_Cam_Logique_Rouleaux : REAL := -19.0;
   Stop_Cam_Logique_Rouleaux : REAL := 31.0;
   Tab_Moyennage_Codeur : REAL[200] := ([1] := 47.14, [2] := 46.948, [3] := 46.676, [4] := 46.404, [5] := 45.66, [6] := 45.576, [7] := 44.956, [8] := 45.08, [9] := 45.792, [10] := 45.956, [11] := 46.692, [12] := 46.608, [13] := 47.104, [14] := 47.328, [15] := 47.844, [16] := 47.896, [17] := 47.632, [18] := 47.02, [19] := 47.008, [20] := 46.712, [21] := 46.684, [22] := 46.084, [23] := 45.672, [24] := 45.34, [25] := 45.448, [26] := 45.624, [27] := 45.74, [28] := 45.764, [29] := 45.476, [30] := 46.336, [31] := 46.684, [32] := 47.588, [33] := 47.752, [34] := 47.912, [35] := 47.636, [36] := 47.636, [37] := 47.38, [38] := 47.14, [39] := 46.592, [40] := 46.224, [41] := 45.444, [42] := 45.188, [43] := 45.32, [44] := 45.488, [45] := 45.956, [46] := 45.924, [47] := 46.472, [48] := 46.788, [49] := 47.196, [50] := 47.5, [51] := 47.488, [52] := 47.172, [53] := 47.54, [54] := 47.344, [55] := 47.296, [56] := 46.684, [57] := 46.32, [58] := 46.22, [59] := 45.896, [60] := 45.62,
        [61] := 45.548, [62] := 45.224, [63] := 45.308, [64] := 45.556, [65] := 46.256, [66] := 46.856, [67] := 47.132, [68] := 47.268, [69] := 47.752, [70] := 47.928, [71] := 47.74, [72] := 48.144, [73] := 47.3, [74] := 46.92, [75] := 46.072, [76] := 45.976, [77] := 45.384, [78] := 45.504, [79] := 44.992, [80] := 45.436, [81] := 45.908, [82] := 46.136, [83] := 46.592, [84] := 46.912, [85] := 47.112, [86] := 47.004, [87] := 47.604, [88] := 47.72, [89] := 47.968, [90] := 47.432, [91] := 47.348, [92] := 46.544, [93] := 46.624, [94] := 45.908, [95] := 46.072, [96] := 45.164, [97] := 45.292, [98] := 45.032, [99] := 45.624, [100] := 46.568, [101] := 46.696, [102] := 47.0, [103] := 47.184, [104] := 47.5, [105] := 47.9, [106] := 47.78, [107] := 47.62, [108] := 47.236, [109] := 46.644, [110] := 46.628, [111] := 45.936, [112] := 46.284, [113] := 45.312, [114] := 45.648, [115] := 45.42, [116] := 45.976, [117] := 45.964, [118] := 46.448, [119] := 46.54, [120] := 46.412,
        [121] := 47.112, [122] := 47.512, [123] := 48.02, [124] := 47.688, [125] := 47.636, [126] := 47.372, [127] := 47.16, [128] := 46.592, [129] := 46.464, [130] := 45.928, [131] := 45.716, [132] := 45.016, [133] := 45.06, [134] := 45.436, [135] := 46.168, [136] := 46.308, [137] := 46.776, [138] := 47.064, [139] := 47.2, [140] := 47.792, [141] := 47.94, [142] := 47.696, [143] := 47.108, [144] := 47.18, [145] := 46.608, [146] := 46.688, [147] := 46.06, [148] := 45.284, [149] := 45.544, [150] := 45.584, [151] := 45.572, [152] := 45.808, [153] := 45.7, [154] := 45.676, [155] := 46.128, [156] := 46.704, [157] := 47.444, [158] := 47.772, [159] := 47.564, [160] := 47.732, [161] := 47.628, [162] := 47.264, [163] := 46.912, [164] := 46.384, [165] := 46.372, [166] := 45.492, [167] := 45.432, [168] := 45.204, [169] := 45.508, [170] := 45.54, [171] := 46.112, [172] := 46.48, [173] := 46.92, [174] := 47.26, [175] := 47.552, [176] := 47.54, [177] := 47.412, [178] := 47.492, [179] := 47.432, [180] := 47.448,
        [181] := 46.4, [182] := 46.444, [183] := 45.98, [184] := 45.9, [185] := 45.376, [186] := 45.628, [187] := 45.208, [188] := 45.252, [189] := 45.364);
   Tab_Moyennage_Codeur_Temp : REAL[200] := ([1] := 46.676, [2] := 46.404, [3] := 45.66, [4] := 45.576, [5] := 44.956, [6] := 45.08, [7] := 45.792, [8] := 45.956, [9] := 46.692, [10] := 46.608, [11] := 47.104, [12] := 47.328, [13] := 47.844, [14] := 47.896, [15] := 47.632, [16] := 47.02, [17] := 47.008, [18] := 46.712, [19] := 46.684, [20] := 46.084, [21] := 45.672, [22] := 45.34, [23] := 45.448, [24] := 45.624, [25] := 45.74, [26] := 45.764, [27] := 45.476, [28] := 46.336, [29] := 46.684, [30] := 47.588, [31] := 47.752, [32] := 47.912, [33] := 47.636, [34] := 47.636, [35] := 47.38, [36] := 47.14, [37] := 46.592, [38] := 46.224, [39] := 45.444, [40] := 45.188, [41] := 45.32, [42] := 45.488, [43] := 45.956, [44] := 45.924, [45] := 46.472, [46] := 46.788, [47] := 47.196, [48] := 47.5, [49] := 47.488, [50] := 47.172, [51] := 47.54, [52] := 47.344, [53] := 47.296, [54] := 46.684, [55] := 46.32, [56] := 46.22, [57] := 45.896, [58] := 45.62, [59] := 45.548, [60] := 45.224,
        [61] := 45.308, [62] := 45.556, [63] := 46.256, [64] := 46.856, [65] := 47.132, [66] := 47.268, [67] := 47.752, [68] := 47.928, [69] := 47.74, [70] := 48.144, [71] := 47.3, [72] := 46.92, [73] := 46.072, [74] := 45.976, [75] := 45.384, [76] := 45.504, [77] := 44.992, [78] := 45.436, [79] := 45.908, [80] := 46.136, [81] := 46.592, [82] := 46.912, [83] := 47.112, [84] := 47.004, [85] := 47.604, [86] := 47.72, [87] := 47.968, [88] := 47.432, [89] := 47.348, [90] := 46.544, [91] := 46.624, [92] := 45.908, [93] := 46.072, [94] := 45.164, [95] := 45.292, [96] := 45.032, [97] := 45.624, [98] := 46.568, [99] := 46.696, [100] := 47.0, [101] := 47.184, [102] := 47.5, [103] := 47.9, [104] := 47.78, [105] := 47.62, [106] := 47.236, [107] := 46.644, [108] := 46.628, [109] := 45.936, [110] := 46.284, [111] := 45.312, [112] := 45.648, [113] := 45.42, [114] := 45.976, [115] := 45.964, [116] := 46.448, [117] := 46.54, [118] := 46.412, [119] := 47.112, [120] := 47.512,
        [121] := 48.02, [122] := 47.688, [123] := 47.636, [124] := 47.372, [125] := 47.16, [126] := 46.592, [127] := 46.464, [128] := 45.928, [129] := 45.716, [130] := 45.016, [131] := 45.06, [132] := 45.436, [133] := 46.168, [134] := 46.308, [135] := 46.776, [136] := 47.064, [137] := 47.2, [138] := 47.792, [139] := 47.94, [140] := 47.696, [141] := 47.108, [142] := 47.18, [143] := 46.608, [144] := 46.688, [145] := 46.06, [146] := 45.284, [147] := 45.544, [148] := 45.584, [149] := 45.572, [150] := 45.808, [151] := 45.7, [152] := 45.676, [153] := 46.128, [154] := 46.704, [155] := 47.444, [156] := 47.772, [157] := 47.564, [158] := 47.732, [159] := 47.628, [160] := 47.264, [161] := 46.912, [162] := 46.384, [163] := 46.372, [164] := 45.492, [165] := 45.432, [166] := 45.204, [167] := 45.508, [168] := 45.54, [169] := 46.112, [170] := 46.48, [171] := 46.92, [172] := 47.26, [173] := 47.552, [174] := 47.54, [175] := 47.412, [176] := 47.492, [177] := 47.432, [178] := 47.448, [179] := 46.4, [180] := 46.444,
        [181] := 45.98, [182] := 45.9, [183] := 45.376, [184] := 45.628, [185] := 45.208, [186] := 45.252, [187] := 45.364, [188] := 45.972, [189] := 46.952, [190] := 47.148);
   Tab_Position_Correction : REAL[50] := ([1] := 59.0, [2] := 59.0, [3] := 59.0, [4] := 59.0, [5] := 59.0, [6] := 59.0, [7] := 59.0, [8] := 59.0, [9] := 59.0, [10] := 59.0, [11] := 59.0, [12] := 59.0, [13] := 59.0, [14] := 59.0, [15] := 59.0, [16] := 59.0, [17] := 59.0, [18] := 59.0, [19] := 59.0, [20] := 59.0, [21] := 59.0, [22] := 59.0, [23] := 59.0, [24] := 59.0, [25] := 59.0, [26] := 59.0, [27] := 59.0, [28] := 59.0, [29] := 59.0, [30] := 59.0, [31] := 59.0, [32] := 30.0, [33] := 30.0, [34] := 30.0, [35] := 30.0, [36] := 30.0, [37] := 30.0, [38] := 30.0, [39] := 30.0);
   Tab_Position_Correction_Temp : REAL[50] := ([1] := 59.0, [2] := 59.0, [3] := 59.0, [4] := 59.0, [5] := 59.0, [6] := 59.0, [7] := 59.0, [8] := 59.0, [9] := 59.0, [10] := 59.0, [11] := 59.0, [12] := 59.0, [13] := 59.0, [14] := 59.0, [15] := 59.0, [16] := 59.0, [17] := 59.0, [18] := 59.0, [19] := 59.0, [20] := 59.0, [21] := 59.0, [22] := 59.0, [23] := 59.0, [24] := 59.0, [25] := 59.0, [26] := 59.0, [27] := 59.0, [28] := 59.0, [29] := 59.0, [30] := 59.0, [31] := 59.0, [32] := 30.0, [33] := 30.0, [34] := 30.0, [35] := 30.0, [36] := 30.0, [37] := 30.0, [38] := 30.0, [39] := 30.0, [40] := 30.0);
   Tableau_Presence_Produit : UDT_REGISTRE_TAPIS[200] := ([1].Position := 10000.0, [1].Etat_Produit := 7, [2].Position := 10000.0, [2].Etat_Produit := 7, [3].Position := 10000.0, [3].Etat_Produit := 7, [4].Position := 10000.0, [4].Etat_Produit := 7, [5].Position := 10000.0, [5].Etat_Produit := 7, [6].Position := 10000.0, [6].Etat_Produit := 7, [7].Position := 10000.0, [7].Etat_Produit := 7, [8].Position := 10000.0, [8].Etat_Produit := 7, [9].Position := 10000.0, [9].Etat_Produit := 7, [10].Position := 10000.0, [10].Etat_Produit := 7, [11].Position := 10000.0, [11].Etat_Produit := 7, [12].Position := 10000.0, [12].Etat_Produit := 7, [13].Position := 10000.0, [13].Etat_Produit := 7, [14].Position := 10000.0, [14].Etat_Produit := 7, [15].Position := 10000.0, [15].Etat_Produit := 7, [16].Position := 10000.0, [16].Etat_Produit := 7, [17].Position := 10000.0, [17].Etat_Produit := 7, [18].Position := 10000.0, [18].Etat_Produit := 7, [19].Position := 10000.0, [19].Etat_Produit := 7, [20].Position := 10000.0, [20].Etat_Produit := 7, [21].Position := 10000.0, [21].Etat_Produit := 7, [22].Position := 10000.0, [22].Etat_Produit := 7, [23].Position := 10000.0, [23].Etat_Produit := 7, [24].Position := 10000.0, [24].Etat_Produit := 7, [25].Position := 10000.0, [25].Etat_Produit := 7, [26].Position := 10000.0, [26].Etat_Produit := 7, [27].Position := 10000.0, [27].Etat_Produit := 7, [28].Position := 10000.0, [28].Etat_Produit := 7, [29].Position := 10000.0, [29].Etat_Produit := 7, [30].Position := 10000.0, [30].Etat_Produit := 7,
        [31].Position := 10000.0, [31].Etat_Produit := 7, [32].Position := 10000.0, [32].Etat_Produit := 7, [33].Position := 10000.0, [33].Etat_Produit := 7, [34].Position := 10000.0, [34].Etat_Produit := 7, [35].Position := 10000.0, [35].Etat_Produit := 7, [36].Position := 10000.0, [36].Etat_Produit := 7, [37].Position := 10000.0, [37].Etat_Produit := 7, [38].Position := 10000.0, [38].Etat_Produit := 7, [39].Position := 10000.0, [39].Etat_Produit := 7, [40].Position := 10000.0, [40].Etat_Produit := 7, [41].Position := 10000.0, [41].Etat_Produit := 7, [42].Position := 10000.0, [42].Etat_Produit := 7, [43].Position := 10000.0, [43].Etat_Produit := 7, [44].Position := 10000.0, [44].Etat_Produit := 7, [45].Position := 10000.0, [45].Etat_Produit := 7, [46].Position := 10000.0, [46].Etat_Produit := 7, [47].Position := 10000.0, [47].Etat_Produit := 7, [48].Position := 10000.0, [48].Etat_Produit := 7, [49].Position := 10000.0, [49].Etat_Produit := 7, [50].Position := 10000.0, [50].Etat_Produit := 7, [51].Position := 10000.0, [51].Etat_Produit := 7, [52].Position := 10000.0, [52].Etat_Produit := 7, [53].Position := 10000.0, [53].Etat_Produit := 7, [54].Position := 10000.0, [54].Etat_Produit := 7, [55].Position := 10000.0, [55].Etat_Produit := 7, [56].Position := 10000.0, [56].Etat_Produit := 7, [57].Position := 10000.0, [57].Etat_Produit := 7, [58].Position := 10000.0, [58].Etat_Produit := 7, [59].Position := 10000.0, [59].Etat_Produit := 7, [60].Position := 10000.0, [60].Etat_Produit := 7,
        [61].Position := 10000.0, [61].Etat_Produit := 7, [62].Position := 10000.0, [62].Etat_Produit := 7, [63].Position := 10000.0, [63].Etat_Produit := 7, [64].Position := 10000.0, [64].Etat_Produit := 7, [65].Position := 10000.0, [65].Etat_Produit := 7, [66].Position := 10000.0, [66].Etat_Produit := 7, [67].Position := 10000.0, [67].Etat_Produit := 7, [68].Position := 10000.0, [68].Etat_Produit := 7, [69].Position := 10000.0, [69].Etat_Produit := 7, [70].Position := 10000.0, [70].Etat_Produit := 7, [71].Position := 10000.0, [71].Etat_Produit := 7, [72].Position := 10000.0, [72].Etat_Produit := 7, [73].Position := 10000.0, [73].Etat_Produit := 7, [74].Position := 10000.0, [74].Etat_Produit := 7, [75].Position := 10000.0, [75].Etat_Produit := 7, [76].Position := 10000.0, [76].Etat_Produit := 7, [77].Position := 10000.0, [77].Etat_Produit := 7, [78].Position := 10000.0, [78].Etat_Produit := 7, [79].Position := 10000.0, [79].Etat_Produit := 7, [80].Position := 10000.0, [80].Etat_Produit := 7, [81].Position := 10000.0, [81].Etat_Produit := 7, [82].Position := 10000.0, [82].Etat_Produit := 7, [83].Position := 10000.0, [83].Etat_Produit := 7, [84].Position := 10000.0, [84].Etat_Produit := 7, [85].Position := 10000.0, [85].Etat_Produit := 7, [86].Position := 10000.0, [86].Etat_Produit := 7, [87].Position := 10000.0, [87].Etat_Produit := 7, [88].Position := 10000.0, [88].Etat_Produit := 7, [89].Position := 10000.0, [89].Etat_Produit := 7, [90].Position := 10000.0, [90].Etat_Produit := 7,
        [91].Position := 10000.0, [91].Etat_Produit := 7, [92].Position := 10000.0, [92].Etat_Produit := 7, [93].Position := 10000.0, [93].Etat_Produit := 7, [94].Position := 10000.0, [94].Etat_Produit := 7, [95].Position := 10000.0, [95].Etat_Produit := 7, [96].Position := 10000.0, [96].Etat_Produit := 7, [97].Position := 10000.0, [97].Etat_Produit := 7, [98].Position := 10000.0, [98].Etat_Produit := 7, [99].Position := 10000.0, [99].Etat_Produit := 7, [100].Position := 10000.0, [100].Etat_Produit := 7, [101].Position := 10000.0, [102].Position := 10000.0, [103].Position := 10000.0, [104].Position := 10000.0, [105].Position := 10000.0, [106].Position := 10000.0, [107].Position := 10000.0, [108].Position := 10000.0, [109].Position := 10000.0, [110].Position := 10000.0, [111].Position := 10000.0, [112].Position := 10000.0, [113].Position := 10000.0, [114].Position := 10000.0, [115].Position := 10000.0, [116].Position := 10000.0, [117].Position := 10000.0, [118].Position := 10000.0, [119].Position := 10000.0, [120].Position := 10000.0, [121].Position := 10000.0, [122].Position := 10000.0, [123].Position := 10000.0, [124].Position := 10000.0, [125].Position := 10000.0, [126].Position := 10000.0, [127].Position := 10000.0, [128].Position := 10000.0, [129].Position := 10000.0, [130].Position := 10000.0, [131].Position := 10000.0, [132].Position := 10000.0, [133].Position := 10000.0, [134].Position := 10000.0, [135].Position := 10000.0, [136].Position := 10000.0, [137].Position := 10000.0, [138].Position := 10000.0, [139].Position := 10000.0, [140].Position := 10000.0,
        [141].Position := 10000.0, [142].Position := 10000.0, [143].Position := 10000.0, [144].Position := 10000.0, [145].Position := 10000.0, [146].Position := 10000.0, [147].Position := 10000.0, [148].Position := 10000.0, [149].Position := 10000.0, [150].Position := 10000.0, [151].Position := 10000.0, [152].Position := 10000.0, [153].Position := 10000.0, [154].Position := 10000.0, [155].Position := 10000.0, [156].Position := 10000.0, [157].Position := 10000.0, [158].Position := 10000.0, [159].Position := 10000.0, [160].Position := 10000.0, [161].Position := 10000.0, [162].Position := 10000.0, [163].Position := 10000.0, [164].Position := 10000.0, [165].Position := 10000.0, [166].Position := 10000.0, [167].Position := 10000.0, [168].Position := 10000.0, [169].Position := 10000.0, [170].Position := 10000.0, [171].Position := 10000.0, [172].Position := 10000.0, [173].Position := 10000.0, [174].Position := 10000.0, [175].Position := 10000.0, [176].Position := 10000.0, [177].Position := 10000.0, [178].Position := 10000.0, [179].Position := 10000.0, [180].Position := 10000.0, [181].Position := 10000.0, [182].Position := 10000.0, [183].Position := 10000.0, [184].Position := 10000.0, [185].Position := 10000.0, [186].Position := 10000.0, [187].Position := 10000.0, [188].Position := 10000.0, [189].Position := 10000.0, [190].Position := 10000.0);
   Tempo_Off_Arret_Rouleaux : TIMER := (PRE := 500, ACC := 475, TT := 1, DN := 1);
   Tempo_RAZ_Ton_Once : TIMER := (PRE := 100);
   tempo_test_tof : TIMER := (PRE := 150, ACC := 150);
   Tempo_Top_Once : FBD_TIMER := (PRE := 100, Reset := 1, ACC := 100);
   Temporisation_Engagement_Virtuel_CF : TIMER := (PRE := 500);
   Temps_total_avant_arret_L4 : REAL := 1000002.0;
   test_arret : BOOL;
   Test_Coupe_Fil : Test_Axe_Avec_Autorisation := (Vitesse := 60.0, Acc := 3600.0, Dec := 3600.0, Jerk := 100.0);
   Test_Coupe_Fil_EN : BOOL;
   Test_Horizontal_Droit : Test_Axe_Avec_Autorisation := (Vitesse := 2.0, Acc := 10.0, Dec := 10.0, Jerk := 100.0, ER := 1);
   Test_Horizontal_Droit_EN : BOOL;
   Test_Horizontal_Gauche : Test_Axe_Avec_Autorisation := (Vitesse := 2.0, Acc := 10.0, Dec := 10.0, Jerk := 100.0, ER := 1);
   Test_Horizontal_Gauche_EN : BOOL;
   Test_Pompe_Doseuse : Test_Axe_Avec_Autorisation := (Vitesse := 0.16666667, Acc := 10.0, Dec := 10.0, Jerk := 100.0);
   Test_Pompe_Doseuse_EN : BOOL;
   Test_Rouleaux_Canneles : Test_Axe_Avec_Autorisation := (Vitesse := 0.16666667, Acc := 10.0, Dec := 10.0, Jerk := 100.0);
   Test_Rouleaux_Canneles_EN : BOOL;
   Test_Vertical_Droit : Test_Axe_Avec_Autorisation := (Vitesse := 2.0, Acc := 10.0, Dec := 10.0, Jerk := 100.0, ER := 1);
   Test_Vertical_Droit_EN : BOOL;
   Test_Vertical_Gauche : Test_Axe_Avec_Autorisation := (Vitesse := 2.0, Acc := 10.0, Dec := 10.0, Jerk := 100.0, ER := 1);
   Test_Vertical_Gauche_EN : BOOL;
   testacquit : BOOL;
   TimeOutResynch_Codeur : TIMER := (PRE := 10000);
   TON_Simul_Produit : TIMER := (PRE := 2546, ACC := 890, EN := 1, TT := 1);
   Val_Position_Recalage : REAL;
   Val_Position_Recalage_Tab1 : REAL := 1.0;
   Val_Position_Recalage_Tab2 : REAL := 4.0;
   Val_Position_Recalage_Tab3 : REAL := 3.0;
   Val_Position_Recalage_Tab4 : REAL := 2.0;
   Val_Position_Recalage_Tab5 : REAL := 2.0;
   Valeur_de_Recalage_Moyennee : REAL;
   Vitesse_Codeur : REAL := 46.128;
   Vitesse_Four4_Real : REAL := 2.7826087;
   Vitesse_Mini_Coupe_Fil : REAL := 192.0;
   Vitesse_Moy_Codeur : REAL := 46.519257;
   Vitesse_Moy_Temp : REAL := 6977.8887;
END_VAR
